// TwinCAT 3 PLC project Fraktal_Press_Demo
// Title: Fraktal_Press_Demo
// Company: fraktal-automation
// Author: fraktal-automation
// ProjectVersion: 0.1.0.7
// Description: CX2030 virtual/physical commissioning example: XTI-linked EK1200/EL1809/EL2809 HAL mapping, two-hand start, interlocked door/part slide, safety aliases, Control On/Off, AUTO/HOME/MANUAL, and model recipes.
// ProgramVersion: 3.1.4024.0
// libraries:
//   Tc2_Standard, * (Beckhoff Automation GmbH)
//   Tc3_Module, * (Beckhoff Automation GmbH)
//   Fraktal_Core, 0.1.0.3 (fraktal-automation)
//   Fraktal_Modules, 0.1.0.2 (fraktal-automation)
// project tree:
//   / PlcTask.TcTTO
//   01_PneumaticPress/Sequences/ FB_PressDemoLoadPosition.TcPOU, FB_PressDemoHome.TcPOU, FB_PressDemoChangeover.TcPOU, FB_PressDemoAuto.TcPOU
//   01_PneumaticPress/Release/ FB_PressDemoRelease.TcPOU
//   01_PneumaticPress/ FB_PressDemoUnit.TcPOU
//   00_System/ MAIN.TcPOU, GVL_PressIO.TcGVL, GVL_PressSafety.TcGVL, FB_PressIoDriver.TcPOU, FB_PressControlDomain.TcPOU, FB_PressOutputAuthority.TcPOU, FB_PressSimulationDriver.TcPOU
//   01_PneumaticPress/Recipes/ FB_PressRecipeCatalog.TcPOU
//   01_PneumaticPress/Io/ FB_PressIoCatalog.TcPOU, GVL_PressFieldbus.TcGVL

CONFIGURATION Fraktal_Press_Demo
    RESOURCE PLC ON TwinCAT3
        TASK PlcTask(INTERVAL := T#10ms, PRIORITY := 20);
        PROGRAM MAIN WITH PlcTask : MAIN;
    END_RESOURCE
END_CONFIGURATION

// ---- 00_System/GVL_PressIO.TcGVL
{attribute 'qualified_only'}
// CX2030 local EtherCAT process image, reconciled with the supplied XTI export.
// TcLinkTo owns the physical link by exact terminal/channel/PDO-entry name;
// AT %I*/%Q* keeps the compiler-selected process-image offset non-positional.
VAR_GLOBAL
    // =000+S-K010B1 (EL1809) inputs
    {attribute 'TcLinkTo' := 'TIIB[=000+S-K010B1 (EL1809)]^Channel 1^_101B301A'}
    _101B301A AT %I* : BOOL;       // Ch1 feeder retracted = logical slide INSIDE
    {attribute 'TcLinkTo' := 'TIIB[=000+S-K010B1 (EL1809)]^Channel 2^_101B301B'}
    _101B301B AT %I* : BOOL;       // Ch2 feeder extended  = logical slide OUTSIDE
    {attribute 'TcLinkTo' := 'TIIB[=000+S-K010B1 (EL1809)]^Channel 3^_101B201A'}
    _101B201A AT %I* : BOOL;       // Ch3 door closed
    {attribute 'TcLinkTo' := 'TIIB[=000+S-K010B1 (EL1809)]^Channel 4^_101B201B'}
    _101B201B AT %I* : BOOL;       // Ch4 door open
    {attribute 'TcLinkTo' := 'TIIB[=000+S-K010B1 (EL1809)]^Channel 5^_101B202A'}
    _101B202A AT %I* : BOOL;       // Ch5 press down
    {attribute 'TcLinkTo' := 'TIIB[=000+S-K010B1 (EL1809)]^Channel 6^_101B202B'}
    _101B202B AT %I* : BOOL;       // Ch6 press up
    {attribute 'TcLinkTo' := 'TIIB[=000+S-K010B1 (EL1809)]^Channel 7^_101S101'}
    _101S101  AT %I* : BOOL;       // Ch7 right two-hand raw button
    {attribute 'TcLinkTo' := 'TIIB[=000+S-K010B1 (EL1809)]^Channel 8^_101S102'}
    _101S102  AT %I* : BOOL;       // Ch8 left two-hand raw button
    {attribute 'TcLinkTo' := 'TIIB[=000+S-K010B1 (EL1809)]^Channel 10^_000MB085A_2'}
    _000MB085A_2 AT %I* : BOOL;    // Ch10 compressed air below 0.3 bar
    {attribute 'TcLinkTo' := 'TIIB[=000+S-K010B1 (EL1809)]^Channel 11^_000MB085A_4'}
    _000MB085A_4 AT %I* : BOOL;    // Ch11 compressed air above 4.5 bar
    {attribute 'TcLinkTo' := 'TIIB[=000+S-K010B1 (EL1809)]^Channel 12^_101B601'}
    _101B601 AT %I* : BOOL;        // Ch12 part present
    {attribute 'TcLinkTo' := 'TIIB[=000+S-K010B1 (EL1809)]^Channel 14^_000K911_Y32'}
    _000K911_Y32 AT %I* : BOOL;    // Ch14 Control On feedback
    {attribute 'TcLinkTo' := 'TIIB[=000+S-K010B1 (EL1809)]^Channel 15^_000K910A'}
    _000K910A AT %I* : BOOL;       // Ch15 ordinary E-stop healthy mirror only

    // =000+S-K010C1 (EL2809) outputs
    {attribute 'TcLinkTo' := 'TIIB[=000+S-K010C1 (EL2809)]^Channel 1^_101K301A'}
    _101K301A AT %Q* : BOOL;       // Ch1 feeder backward = move inside
    {attribute 'TcLinkTo' := 'TIIB[=000+S-K010C1 (EL2809)]^Channel 2^_101K301B'}
    _101K301B AT %Q* : BOOL;       // Ch2 feeder forward  = move outside
    {attribute 'TcLinkTo' := 'TIIB[=000+S-K010C1 (EL2809)]^Channel 3^_101K201A'}
    _101K201A AT %Q* : BOOL;       // Ch3 close door
    {attribute 'TcLinkTo' := 'TIIB[=000+S-K010C1 (EL2809)]^Channel 4^_101K201B'}
    _101K201B AT %Q* : BOOL;       // Ch4 open door
    {attribute 'TcLinkTo' := 'TIIB[=000+S-K010C1 (EL2809)]^Channel 5^_101K202A'}
    _101K202A AT %Q* : BOOL;       // Ch5 press downward
    {attribute 'TcLinkTo' := 'TIIB[=000+S-K010C1 (EL2809)]^Channel 6^_101K202B'}
    _101K202B AT %Q* : BOOL;       // Ch6 press upward
    {attribute 'TcLinkTo' := 'TIIB[=000+S-K010C1 (EL2809)]^Channel 7^_101P101'}
    _101P101  AT %Q* : BOOL;       // Ch7 right two-hand lamp
    {attribute 'TcLinkTo' := 'TIIB[=000+S-K010C1 (EL2809)]^Channel 8^_101P102'}
    _101P102  AT %Q* : BOOL;       // Ch8 left two-hand lamp
    {attribute 'TcLinkTo' := 'TIIB[=000+S-K010C1 (EL2809)]^Channel 10^_000K951_A1'}
    _000K951_A1 AT %Q* : BOOL;     // Ch10 SwitchControlOn functional request
    {attribute 'TcLinkTo' := 'TIIB[=000+S-K010C1 (EL2809)]^Channel 11^_000K911_A1'}
    _000K911_A1 AT %Q* : BOOL;     // Ch11 EnableControlOn functional request
END_VAR

// ---- 00_System/GVL_PressSafety.TcGVL
{attribute 'qualified_only'}
// Read-only aliases to results produced outside the standard PLC by TwinSAFE
// or a validated external safety system. They intentionally default FALSE so
// physical mode cannot energize until commissioning supplies every result.
// These variables do not themselves implement a safety function.
VAR_GLOBAL
    _EStopOk               AT %I* : BOOL;
    _GuardClosed           AT %I* : BOOL;
    _TwoHandActive         AT %I* : BOOL;
    _PneumaticPermit       AT %I* : BOOL;
    _SafetyFieldbusHealthy AT %I* : BOOL;
    _StandardIoHealthy     AT %I* : BOOL;
END_VAR

// ---- 01_PneumaticPress/Io/GVL_PressFieldbus.TcGVL
{attribute 'qualified_only'}
{attribute 'OPC.UA.DA' := '1'}
// Owner-local, bounded publication of the demo's physical CX2030 I/O tree.
// ST_IoChannel.Name is always the exact electrical-list/schematic tag.
VAR_GLOBAL
    Topology : ST_FieldbusTopology;
END_VAR

// ---- 00_System/MAIN.TcPOU
// Virtual-commissioning application for one pneumatic press Unit.
// IMPORTANT: the Safe* values below simulate TwinSAFE outputs only. A deployed
// machine maps certified E-stop/two-hand/guard/safe-valve results from TwinSAFE.
PROGRAM MAIN
VAR
    RecipeCatalog : FB_PressRecipeCatalog;
    PartCarrier : FB_LocalPartCarrier;    // §3.16.2 BY_POSITION identity + local result ring
    AccessUsers : FB_LocalAccessProvider; // §7.7 commissioning user/PIN table
    // TF6100 TMC-Filtered publication starts at the deployed root instance.
    // The marker is inherited by PneumaticPress's published child symbols.
    {attribute 'OPC.UA.DA' := '1'}
    PneumaticPress : FB_PressDemoUnit;
    IoCatalog : FB_PressIoCatalog;
    IoDriver : FB_PressIoDriver;
    ControlDomain : FB_PressControlDomain;
    OutputAuthority : FB_PressOutputAuthority;
    SimulationDriver : FB_PressSimulationDriver;
    PressHal, DoorHal, SlideHal : ST_CylinderHal;
    TwoHandHal : ST_TwoHandHal;
    PowerHal : ST_PowerGroupHal;
    PartPresentHal : ST_DigitalInputHal;
    AirPressureHal : ST_AirPressureHal;
    InitialModel : ST_ModelId;
    Plate : ST_Nameplate;
    Init : BOOL;
    UseSimulation : BOOL := TRUE; // set FALSE only after I/O + safety aliases are linked
    ControlCircuitMappingConfirmed : BOOL; // verify K951/K911 electrical semantics first

    // Simulation controls. E-stop is normally closed: TRUE = healthy circuit.
    SimEStopNc : BOOL := TRUE;
    SimControlOnButton : BOOL;
    SimControlOffButton : BOOL;
    SimLeftButton : BOOL;
    SimRightButton : BOOL;
    SimSafetyValveOk : BOOL := TRUE;
    SimFieldbusHealthy : BOOL := TRUE;
    SimPartPresent : BOOL := TRUE;
    SimAirPressureOk : BOOL := TRUE;
    SafeEStopOk : BOOL;
    SafeGuardClosed : BOOL;
    SafeTwoHandActive : BOOL;
    SafePneumaticPermit : BOOL;
    SafetyFieldbusHealthy : BOOL;
    StandardIoHealthy : BOOL;
    RawEStopHealthy : BOOL;
    LampsOn : BOOL;
    ControlOnEdge : R_TRIG;
    ControlOffEdge : R_TRIG;
END_VAR

IF NOT Init THEN
    Init := TRUE;
    // Initial mechanically safe/load position: ram up, door open, slide outside.
    PressHal.RetractedFb := TRUE;
    DoorHal.RetractedFb := TRUE;
    SlideHal.RetractedFb := TRUE;
    RecipeCatalog.Setup(UnitRef := PneumaticPress);
    PneumaticPress.Setup(Name := 'PneumaticPress', PressHal := PressHal, DoorHal := DoorHal,
        SlideHal := SlideHal, TwoHandHal := TwoHandHal, PowerHal := PowerHal,
        PartPresentHal := PartPresentHal, AirPressureHal := AirPressureHal,
        Recipe := RecipeCatalog.Provider);
    IoDriver.Setup(UnitRef := PneumaticPress);
    IoCatalog.Setup(UnitRef := PneumaticPress);
    ControlDomain.Setup(UnitRef := PneumaticPress);
    SimulationDriver.Setup(PressHal := PressHal, DoorHal := DoorHal, SlideHal := SlideHal);
    InitialModel.ModelCode := 'ALUMINUM';
    PneumaticPress.SetModel(Id := InitialModel);
    Plate.ProductUri := 'urn:fraktal:demo:pneumatic-press:2026-0001';
    Plate.ManufacturerName := 'Fraktal Example Project';
    Plate.ProductDesignation := 'Pneumatic Press Training Cell';
    Plate.SerialNumber := 'PRESS-DEMO-2026-0001';
    Plate.YearOfConstruction := '2026';
    Plate.SoftwareVersion := 'Fraktal Press Demo 0.1';
    PneumaticPress.SetNameplate(Plate := Plate);
    PneumaticPress.AlarmLog.RegisterMeta(Reason := E_Reason.INTERLOCK_DROPPED,
        OperatorAction := 'project.alarmAction.pressInterlock',
        Consequence := 'project.alarmConsequence.pressInterlock', Shelvable := FALSE);
    // §8.9 rationalization: per-reason operator action + consequence for the HMI join
    PneumaticPress.AlarmLog.RegisterMeta(Reason := E_Reason.PERMISSIVE_NOT_MET,
        OperatorAction := 'project.alarmAction.pressAirPressure',
        Consequence := 'project.alarmConsequence.pressAirPressure', Shelvable := FALSE);
    PneumaticPress.AlarmLog.RegisterMeta(Reason := E_Reason.RECIPE_INVALID,
        OperatorAction := 'project.alarmAction.pressRecipe',
        Consequence := 'project.alarmConsequence.pressRecipe', Shelvable := FALSE);
    PneumaticPress.AlarmLog.RegisterMeta(Reason := PL_ModuleReasons.CYL_WORK_NOT_REACHED,
        OperatorAction := 'project.alarmAction.pressCylinderPosition',
        Consequence := 'project.alarmConsequence.pressCylinderPosition', Shelvable := FALSE);
    PneumaticPress.AlarmLog.RegisterMeta(Reason := PL_ModuleReasons.CYL_HOME_NOT_REACHED,
        OperatorAction := 'project.alarmAction.pressCylinderPosition',
        Consequence := 'project.alarmConsequence.pressCylinderPosition', Shelvable := FALSE);
    // §3.16 traceability: station-local BY_POSITION serials; RFID/host substitutes later
    PartCarrier.Setup(UidPrefix := 'PRESS-2026-');
    PneumaticPress.SetPartCarrier(Carrier := PartCarrier);
    // §7.7 access: commissioning users (policy stays shipped-open; login is optional)
    AccessUsers.Register(User := 'operator', Pin := '1111', Level := E_AccessLevel.OPERATOR);
    AccessUsers.Register(User := 'tech', Pin := '2222', Level := E_AccessLevel.TECHNICIAN);
    AccessUsers.Register(User := 'admin', Pin := '9999', Level := E_AccessLevel.ADMIN);
    PneumaticPress.Access.Setup(Provider := AccessUsers, pAlarmLog := ADR(PneumaticPress.AlarmLog));
END_IF

// Ordinary simulated local station buttons. The worksheet does not list real
// Control On/Off input buttons; physical operation therefore uses HMI requests
// until those devices are identified. Control Off wins simultaneous edges.
ControlOnEdge(CLK := UseSimulation AND SimControlOnButton);
ControlOffEdge(CLK := UseSimulation AND SimControlOffButton);
IF ControlOffEdge.Q THEN
    PneumaticPress.RequestLocalControl(ControlOn := FALSE);
ELSIF ControlOnEdge.Q THEN
    PneumaticPress.RequestLocalControl(ControlOn := TRUE);
END_IF

IF UseSimulation THEN
    SimulationDriver.M_ReadInputs(DoorHal := DoorHal, TwoHandHal := TwoHandHal,
        PowerHal := PowerHal, PartPresentHal := PartPresentHal,
        AirPressureHal := AirPressureHal, RawEStopHealthy := RawEStopHealthy,
        SafeEStopOk := SafeEStopOk, SafeGuardClosed := SafeGuardClosed,
        SafeTwoHandActive := SafeTwoHandActive,
        SafePneumaticPermit := SafePneumaticPermit,
        SafetyFieldbusHealthy := SafetyFieldbusHealthy,
        StandardIoHealthy := StandardIoHealthy, SimEStopNc := SimEStopNc,
        SimLeftButton := SimLeftButton, SimRightButton := SimRightButton,
        SimSafetyValveOk := SimSafetyValveOk,
        SimFieldbusHealthy := SimFieldbusHealthy,
        SimPartPresent := SimPartPresent, SimAirPressureOk := SimAirPressureOk,
        PowerRequested := PowerHal.EnableRequestOut);
ELSE
    // The project Hardware Driver is the only raw process-image consumer.
    IoDriver.M_ReadInputs(PressHal := PressHal, DoorHal := DoorHal,
        SlideHal := SlideHal, TwoHandHal := TwoHandHal, PowerHal := PowerHal,
        PartPresentHal := PartPresentHal, AirPressureHal := AirPressureHal,
        RawEStopHealthy := RawEStopHealthy, SafeEStopOk := SafeEStopOk,
        SafeGuardClosed := SafeGuardClosed, SafeTwoHandActive := SafeTwoHandActive,
        SafePneumaticPermit := SafePneumaticPermit,
        SafetyFieldbusHealthy := SafetyFieldbusHealthy,
        StandardIoHealthy := StandardIoHealthy);
END_IF
TwoHandHal.SafeActive := SafeTwoHandActive;
TwoHandHal.FieldbusHealthy := SafetyFieldbusHealthy;
PowerHal.SafetyPermit := SafePneumaticPermit;
PowerHal.FieldbusHealthy := StandardIoHealthy;

ControlDomain.M_Update(SafeEStopOk := SafeEStopOk,
    SafeGuardClosed := SafeGuardClosed, SafeTwoHandActive := SafeTwoHandActive,
    SafePneumaticPermit := SafePneumaticPermit,
    SafetyFieldbusHealthy := SafetyFieldbusHealthy,
    StandardIoHealthy := StandardIoHealthy, RawEStopHealthy := RawEStopHealthy,
    PowerFeedback := PowerHal.PowerFeedback,
    PowerRequested := PowerHal.EnableRequestOut,
    TwoHandFieldbusHealthy := TwoHandHal.FieldbusHealthy);
PneumaticPress.ControlDomain := ControlDomain.Status;

// First execute ordinary control, then apply a standard-PLC withdrawal layer.
// This is defense in depth only: the real safety system owns pneumatic removal.
PneumaticPress();
OutputAuthority.M_Apply(PressHal := PressHal, DoorHal := DoorHal,
    SlideHal := SlideHal, PowerFeedback := PowerHal.PowerFeedback,
    SafePneumaticPermit := SafePneumaticPermit,
    StandardIoHealthy := StandardIoHealthy,
    HazardousRamPermit := SafeGuardClosed AND SafeTwoHandActive);
IF UseSimulation THEN
    // Never leave physical outputs energized while virtual commissioning.
    IoDriver.M_ClearOutputs();
    SimulationDriver.M_RefreshPlant();
ELSE
    LampsOn := PneumaticPress.TwoHand.OutImm.Armed
        AND ControlDomain.Status.ReadyForStart
        AND PneumaticPress.OutImm.PartPresent AND PneumaticPress.OutImm.AirPressureOk;
    IoDriver.M_WriteOutputs(PressHal := PressHal, DoorHal := DoorHal,
        SlideHal := SlideHal, PowerHal := PowerHal, LampsOn := LampsOn,
        ControlCircuitMappingConfirmed := ControlCircuitMappingConfirmed);
END_IF
IoDriver.M_RefreshFieldbus(StandardIoHealthy := StandardIoHealthy);

END_PROGRAM

// ---- 01_PneumaticPress/Recipes/FB_PressRecipeCatalog.TcPOU
// Owner-local recipe engineering data: model identities and their typed Unit records.
// Generic validation/storage remains in FB_LocalRecipeProvider; process behavior
// remains in the project-owned FB_PressDemoUnit. MAIN only composes the two.
FUNCTION_BLOCK FB_PressRecipeCatalog
VAR_OUTPUT
    {attribute 'OPC.UA.DA' := '0'}
    Provider : FB_LocalRecipeProvider;
END_VAR
VAR
    _default : ST_PneumaticPressParCfg;
    _aluminum : ST_PneumaticPressParCfg;
    _plastic : ST_PneumaticPressParCfg;
    _steel : ST_PneumaticPressParCfg;
    _model : ST_ModelId;
    _configured : BOOL;
END_VAR

// Static catalog: no cyclic work.

METHOD Setup : BOOL
VAR_INPUT
    UnitRef : REFERENCE TO FB_PressDemoUnit;
END_VAR
VAR
    Ok : BOOL;
END_VAR
IF _configured THEN
    Setup := TRUE;
    RETURN;
END_IF

// §8.11 per-model performance references: IdealCycleMs feeds OEE Performance
// (§8.5.1); BaselineWorkMs arms the WORK-time degradation watch (§8.11.4(d)).
// Values = design cycle for this training cell (motions + settle + dwell).
_default.PressSettleTime := T#500MS;
_default.TransferSettleTime := T#100MS;
_default.RequireTwoHandStart := TRUE;
_default.IdealCycleMs := 6000;
_default.BaselineWorkMs := 6000;
_aluminum.PressSettleTime := T#300MS;
_aluminum.TransferSettleTime := T#80MS;
_aluminum.RequireTwoHandStart := TRUE;
_aluminum.IdealCycleMs := 5700;
_aluminum.BaselineWorkMs := 5700;
_plastic.PressSettleTime := T#650MS;
_plastic.TransferSettleTime := T#120MS;
_plastic.RequireTwoHandStart := TRUE;
_plastic.IdealCycleMs := 6200;
_plastic.BaselineWorkMs := 6200;
_steel.PressSettleTime := T#1200MS;
_steel.TransferSettleTime := T#150MS;
_steel.RequireTwoHandStart := TRUE;
_steel.IdealCycleMs := 6800;
_steel.BaselineWorkMs := 6800;

Ok := Provider.Register(ModelCode := '', RecipeKey := 'PneumaticPressUnit',
    pData := ADR(_default), Size := SIZEOF(_default));
Ok := Provider.Register(ModelCode := 'ALUMINUM', RecipeKey := 'PneumaticPressUnit',
    pData := ADR(_aluminum), Size := SIZEOF(_aluminum)) AND Ok;
Ok := Provider.Register(ModelCode := 'PLASTIC', RecipeKey := 'PneumaticPressUnit',
    pData := ADR(_plastic), Size := SIZEOF(_plastic)) AND Ok;
Ok := Provider.Register(ModelCode := 'STEEL', RecipeKey := 'PneumaticPressUnit',
    pData := ADR(_steel), Size := SIZEOF(_steel)) AND Ok;

_model.ModelCode := 'ALUMINUM';
Ok := UnitRef.RegisterAvailableModel(Id := _model) AND Ok;
_model.ModelCode := 'PLASTIC';
Ok := UnitRef.RegisterAvailableModel(Id := _model) AND Ok;
_model.ModelCode := 'STEEL';
Ok := UnitRef.RegisterAvailableModel(Id := _model) AND Ok;

_configured := Ok;
Setup := Ok;
END_METHOD

END_FUNCTION_BLOCK

// ---- 01_PneumaticPress/FB_PressDemoUnit.TcPOU
// Project-owned Unit: pneumatic press + access door + transfer slide + two-hand request.
// Cylinder interlocks prevent the two documented collisions in AUTO and MANUAL.
// Certified E-stop, two-hand evaluation and safe valve outputs remain external.
{attribute 'OPC.UA.DA' := '1'}
FUNCTION_BLOCK FB_PressDemoUnit EXTENDS FB_UnitBase
VAR_INPUT
    ParCfg : ST_PneumaticPressParCfg;
    ParCmd : ST_PneumaticPressParCmd;
END_VAR
VAR_OUTPUT
    PressRam      : FB_CylinderCM;
    Door          : FB_CylinderCM;
    PartSlide     : FB_CylinderCM;
    TwoHand       : FB_TwoHandStartCM;
    PneumaticPower: FB_PowerGroupCM;
    PartPresentSensor : FB_DigitalInputCM;
    AirPressureMonitor : FB_AirPressureMonitorCM;
    ReleaseConditions : FB_PressDemoRelease; // project-owned, browseable condition state
    OutCmd        : ST_PneumaticPressOutCmd;
    OutImm        : ST_PneumaticPressOutImm;
END_VAR
VAR
    _recipe : I_RecipeProvider;
    _parCfgStaged : ST_PneumaticPressParCfg;
    _recipePrepared : BOOL;
    _startLatched : BOOL;
    _powerRequestPending : BOOL;
    _powerTargetOn : BOOL;
    {attribute 'OPC.UA.DA' := '0'}
    _homeSequence : FB_PressDemoHome;       // §6.8 ST chain on FB_SequenceBase owns HOME steps
    {attribute 'OPC.UA.DA' := '0'}
    _changeoverSequence : FB_PressDemoChangeover;
    {attribute 'OPC.UA.DA' := '0'}
    _autoSequence : FB_PressDemoAuto;
END_VAR

Cyclic();

METHOD Setup : BOOL
VAR_INPUT
    Name : STRING(80);
    PressHal : REFERENCE TO ST_CylinderHal;
    DoorHal : REFERENCE TO ST_CylinderHal;
    SlideHal : REFERENCE TO ST_CylinderHal;
    TwoHandHal : REFERENCE TO ST_TwoHandHal;
    PowerHal : REFERENCE TO ST_PowerGroupHal;
    PartPresentHal : REFERENCE TO ST_DigitalInputHal;
    AirPressureHal : REFERENCE TO ST_AirPressureHal;
    Recipe : I_RecipeProvider;
END_VAR
VAR
    InitialModel : ST_ModelId;
    Ok : BOOL;
END_VAR
_M_SetName(Name);
_M_SetPresentation(DisplayNameKey := 'project.module.pneumaticPress.name', DescriptionKey := 'project.module.pneumaticPress.description');
_recipe := Recipe;
Ok := PressRam.Setup(Name := CONCAT(Name, '.PressRam'), HalRef := PressHal, Recipe := 0);
Ok := Door.Setup(Name := CONCAT(Name, '.Door'), HalRef := DoorHal, Recipe := 0) AND Ok;
Ok := PartSlide.Setup(Name := CONCAT(Name, '.PartSlide'), HalRef := SlideHal, Recipe := 0) AND Ok;
Ok := TwoHand.Setup(Name := CONCAT(Name, '.TwoHand'), HalRef := TwoHandHal) AND Ok;
Ok := PneumaticPower.Setup(Name := CONCAT(Name, '.PneumaticPower'), HalRef := PowerHal) AND Ok;
Ok := PartPresentSensor.Setup(Name := CONCAT(Name, '.PartPresentSensor'),
    HalRef := PartPresentHal, DisplayNameKey := 'project.module.partPresentSensor.name',
    DescriptionKey := 'project.module.partPresentSensor.description') AND Ok;
Ok := AirPressureMonitor.Setup(Name := CONCAT(Name, '.AirPressureMonitor'),
    HalRef := AirPressureHal) AND Ok;
Ok := ReleaseConditions.Setup(UnitPath := Name) AND Ok;
Ok := _homeSequence.Setup(Host := THIS^, PressRam := PressRam, Door := Door,
    PartSlide := PartSlide, OutCmd := OutCmd) AND Ok;
Ok := _changeoverSequence.Setup(Host := THIS^, PressRam := PressRam, Door := Door,
    PartSlide := PartSlide, OutCmd := OutCmd, Model := Model) AND Ok;
Ok := _autoSequence.Setup(Host := THIS^, PressRam := PressRam, Door := Door,
    PartSlide := PartSlide, TwoHand := TwoHand, PartPresentSensor := PartPresentSensor,
    AirPressureMonitor := AirPressureMonitor, ParCfg := ParCfg, OutCmd := OutCmd,
    StartLatched := _startLatched) AND Ok;
PneumaticPower.ParCfg.Kind := E_PowerGroupKind.VALVE_ZONE;
PneumaticPower.ParCfg.RequiredForControl := TRUE;
PneumaticPower.ParCfg.FieldbusLossReaction := E_FieldbusLossReaction.CONTROL_OFF;
Ok := _M_Register(PressRam) AND Ok;
Ok := _M_Register(Door) AND Ok;
Ok := _M_Register(PartSlide) AND Ok;
Ok := _M_Register(TwoHand) AND Ok;
Ok := _M_Register(PneumaticPower) AND Ok;
Ok := _M_Register(PartPresentSensor) AND Ok;
Ok := _M_Register(AirPressureMonitor) AND Ok;
Setup := Ok AND PrepareRecipe(Model := InitialModel);
IF Setup THEN CommitRecipe(); END_IF
END_METHOD

METHOD PrepareRecipe : BOOL
VAR_INPUT
    Model : ST_ModelId;
END_VAR
IF _recipe = 0 THEN
    _parCfgStaged := ParCfg;
    _recipePrepared := TRUE;
ELSIF _recipe.Load(ModelCode := Model.ModelCode, RecipeKey := 'PneumaticPressUnit', pParCfg := ADR(_parCfgStaged), Size := SIZEOF(_parCfgStaged)) THEN
    IF (_parCfgStaged.PressSettleTime > T#30S) OR (_parCfgStaged.TransferSettleTime > T#5S) THEN
        _M_Fault(E_Reason.RECIPE_INVALID, 'project.error.pressRecipeInvalid');
        _recipePrepared := FALSE;
        PrepareRecipe := FALSE;
        RETURN;
    END_IF
    _recipePrepared := TRUE;
ELSE
    _M_Fault(E_Reason.RECIPE_INVALID, 'std.error.recipeSchemaInvalid');
    _recipePrepared := FALSE;
    PrepareRecipe := FALSE;
    RETURN;
END_IF
PrepareRecipe := SUPER^.PrepareRecipe(Model := Model);
IF NOT PrepareRecipe THEN _recipePrepared := FALSE; END_IF
END_METHOD

METHOD CommitRecipe
SUPER^.CommitRecipe();
IF _recipePrepared THEN
    ParCfg := _parCfgStaged;
    // §8.11 performance references follow the model: OEE Performance denominator
    // and the WORK-time degradation baseline are per-recipe engineering data.
    Oee.IdealCycleMs := ParCfg.IdealCycleMs;
    Profiler.M_SetBaselineWork(WorkMs := ParCfg.BaselineWorkMs);
END_IF
_recipePrepared := FALSE;
END_METHOD

METHOD AbortRecipe
SUPER^.AbortRecipe();
_recipePrepared := FALSE;
END_METHOD

METHOD PROTECTED OnCyclic : DINT
OnCyclic := SUPER^.OnCyclic();
// Project release engineering is a separate visible component. It owns the
// functional collision permits and mode-entry conditions consumed below.
ReleaseConditions.M_Evaluate(PressRam := PressRam, Door := Door, PartSlide := PartSlide,
    TwoHand := TwoHand, PneumaticPower := PneumaticPower,
    AirPressure := AirPressureMonitor);

// Latch access-gated Unit requests, then observe one full Execute-low scan before
// starting another power-group command (PLCopen edge discipline).
IF ControlOffRequest THEN
    _powerTargetOn := FALSE;
    _powerRequestPending := TRUE;
ELSIF ControlOnRequest THEN
    _powerTargetOn := TRUE;
    _powerRequestPending := TRUE;
END_IF
IF PneumaticPower.Done OR PneumaticPower.Error OR PneumaticPower.Aborted THEN
    PneumaticPower.Execute := FALSE;
ELSIF _powerRequestPending AND NOT PneumaticPower.Execute
AND (PneumaticPower.State = E_ExecState.READY) THEN
    PneumaticPower.Abort := FALSE;
    IF _powerTargetOn THEN
        PneumaticPower.Command := E_PowerGroupCommand.POWER_ON;
    ELSE
        PneumaticPower.Command := E_PowerGroupCommand.POWER_OFF;
    END_IF
    PneumaticPower.Execute := TRUE;
    _powerRequestPending := FALSE;
END_IF

// A physical two-hand edge may start AUTO from READY, or release an already
// running Unit's wait step. It never bypasses domain readiness or access policy.
IF TwoHand.OutImm.StartPulse
AND PartPresentSensor.OutImm.Value AND PartPresentSensor.OutImm.Quality
AND AirPressureMonitor.OutImm.PressureOk THEN
    IF (State = E_ExecState.BUSY) AND (ModeActive = E_Mode.AUTO) THEN
        _startLatched := TRUE;
    ELSIF (ModeActive = E_Mode.AUTO) AND Start() THEN
        _startLatched := TRUE;
    END_IF
ELSIF TwoHand.OutImm.StartPulse THEN
    _startLatched := FALSE;
END_IF
IF PneumaticPower.Error AND (State = E_ExecState.BUSY) THEN
    _M_RollupFault();
END_IF
IF (State = E_ExecState.BUSY) AND (_step > 10)
AND NOT AirPressureMonitor.OutImm.PressureOk THEN
    PressRam.WithdrawOutputs();
    Door.WithdrawOutputs();
    PartSlide.WithdrawOutputs();
    _M_Fault(E_Reason.PERMISSIVE_NOT_MET, 'project.error.pressAirPressureLost');
END_IF
OutImm.PressRetracted := PressRam.OutImm.Retracted;
OutImm.DoorOpen := Door.OutImm.Retracted;
OutImm.DoorClosed := Door.OutImm.Extended;
OutImm.SlideInside := PartSlide.OutImm.Extended;
OutImm.SlideOutside := PartSlide.OutImm.Retracted;
OutImm.TwoHandArmed := TwoHand.OutImm.Armed;
OutImm.TwoHandActive := TwoHand.OutImm.SafeActive;
OutImm.PartPresent := PartPresentSensor.OutImm.Value AND PartPresentSensor.OutImm.Quality;
OutImm.AirPressureOk := AirPressureMonitor.OutImm.PressureOk;
OutImm.ReadyForLoad := Door.OutImm.Retracted AND NOT Door.OutImm.Extended
    AND PartSlide.OutImm.Retracted AND NOT PartSlide.OutImm.Extended
    AND PressRam.OutImm.Retracted AND NOT PressRam.OutImm.Extended;
OutImm.ActiveSettleTime := ParCfg.PressSettleTime;
OutImm.Diagnostic := Status.Diagnostic;
END_METHOD

METHOD PROTECTED OnAbort : DINT
OnAbort := SUPER^.OnAbort();
_M_PartAborted();                    // §3.16.3: the part leaves without a valid result
PressRam.WithdrawOutputs();
Door.WithdrawOutputs();
PartSlide.WithdrawOutputs();
PressRam.Execute := FALSE;
Door.Execute := FALSE;
PartSlide.Execute := FALSE;
Decision.Prompt := '';
DecisionAnswer := 0;
_startLatched := FALSE;
_homeSequence.M_Reset();
_changeoverSequence.M_Reset();
_autoSequence.M_Reset();
_powerTargetOn := FALSE;
_powerRequestPending := TRUE;
END_METHOD

// Application-only seam for ordinary hardwired Control On/Off buttons.
// It is a method (not OPC UA data), so HMI writes still use the access-gated
// ReqControlOn/ReqControlOff contract. The power CM rechecks safety and health.
METHOD RequestLocalControl : BOOL
VAR_INPUT
    ControlOn : BOOL;
END_VAR
_powerTargetOn := ControlOn;
_powerRequestPending := TRUE;
RequestLocalControl := TRUE;
END_METHOD

// §3.4.2 — the press paces every motion boundary through _M_StepGate, so
// SINGLE_STEP and HOLD_TO_RUN are supported (NON-SAFETY pacing; interlocks
// and the certified safety layer are unaffected).
METHOD PROTECTED _M_SupportsRunStyle : BOOL
VAR_INPUT
    Style : E_RunStyle;
END_VAR
_M_SupportsRunStyle := (Style = E_RunStyle.CONTINUOUS)
    OR (Style = E_RunStyle.SINGLE_STEP) OR (Style = E_RunStyle.HOLD_TO_RUN);
END_METHOD

METHOD PROTECTED _M_Supports : BOOL
VAR_INPUT
    Mode : E_Mode;
END_VAR
_M_Supports := (Mode = E_Mode.AUTO) OR (Mode = E_Mode.MANUAL)
    OR (Mode = E_Mode.HOME) OR (Mode = E_Mode.CHANGEOVER);
END_METHOD

// Thin mode router. Each supported sequence is a named method in the Unit tree.
METHOD PROTECTED _M_Dispatch
CASE ModeActive OF
    E_Mode.AUTO:
        _M_SequenceAuto();
    E_Mode.HOME:
        _M_SequenceHome();
    E_Mode.CHANGEOVER:
        _M_SequenceChangeover();
    E_Mode.MANUAL:
        _M_Fault(E_Reason.UNSUPPORTED_COMMAND, 'project.error.pressManualHasNoSequence');
ELSE
    _M_Fault(E_Reason.UNSUPPORTED_COMMAND, 'project.error.pressModeHasNoSequence');
END_CASE
END_METHOD

// HOME adapter: reset the chain on the first dispatch scan, then run it each scan.
// The §6.8 ST chain (FB_PressDemoHome) owns all HOME step logic.
METHOD PROTECTED _M_SequenceHome
CASE _step OF
    10:
        _homeSequence.M_Reset();
        _step := 20;
    20:
        _homeSequence.M_Run();
ELSE
    PressRam.WithdrawOutputs();
    Door.WithdrawOutputs();
    PartSlide.WithdrawOutputs();
    _M_Fault(E_Reason.STEP_STALLED, 'std.error.undefinedStep');
END_CASE
END_METHOD

// CHANGEOVER adapter: reset then run. The §6.8 ST chain owns model validation,
// safe positioning, the operator decision, and completion logic.
METHOD PROTECTED _M_SequenceChangeover
CASE _step OF
    10:
        _changeoverSequence.M_Reset();
        _step := 20;
    20:
        _changeoverSequence.M_Run();
ELSE
    PressRam.WithdrawOutputs();
    Door.WithdrawOutputs();
    PartSlide.WithdrawOutputs();
    _M_Fault(E_Reason.STEP_STALLED, 'std.error.undefinedStep');
END_CASE
END_METHOD

// AUTO adapter: reset then run. Every production step's command, wait, timer,
// decision, traceability, and transition logic lives in the §6.8 ST chain.
METHOD PROTECTED _M_SequenceAuto
CASE _step OF
    10:
        _autoSequence.M_Reset();
        _step := 20;
    20:
        _autoSequence.M_Run();
ELSE
    PressRam.WithdrawOutputs();
    Door.WithdrawOutputs();
    PartSlide.WithdrawOutputs();
    _M_Fault(E_Reason.STEP_STALLED, 'std.error.undefinedStep');
END_CASE
END_METHOD

METHOD PROTECTED _M_RouteManual : BOOL
VAR_INPUT
    TargetPath : STRING(255);
    Value : DINT;
END_VAR
_M_RouteManual := FALSE;
IF TargetPath = PressRam.Name THEN
    _M_RouteManual := PressRam.ManualCommand(Value := Value);
ELSIF TargetPath = Door.Name THEN
    _M_RouteManual := Door.ManualCommand(Value := Value);
ELSIF TargetPath = PartSlide.Name THEN
    _M_RouteManual := PartSlide.ManualCommand(Value := Value);
ELSE
    _M_RouteManual := FALSE;
END_IF
END_METHOD

// §7.8 mode-entry release owned by this Unit. The base Start method consumes the
// same report the HMI displays, so this condition cannot become explanation-only.
METHOD PROTECTED _M_AppendInterlocks
VAR_IN_OUT
    Report : ST_ReleaseReport;
END_VAR
ReleaseConditions.M_AppendStart(Report := Report);
END_METHOD

METHOD PROTECTED _M_AppendManualInterlocks
VAR_INPUT
    TargetPath : STRING(255);
    Value : DINT;
END_VAR
VAR_IN_OUT
    Report : ST_ReleaseReport;
END_VAR
ReleaseConditions.M_AppendManual(TargetPath := TargetPath, Value := Value,
    PressRam := PressRam, Door := Door, PartSlide := PartSlide, Report := Report);
END_METHOD

METHOD PROTECTED _M_PublishStatus
SUPER^._M_PublishStatus();
OutImm.Diagnostic := Status.Diagnostic;
END_METHOD

END_FUNCTION_BLOCK

// ---- 01_PneumaticPress/Release/FB_PressDemoRelease.TcPOU
// Project-owned release engineering for the pneumatic press.
// This FB is not a Fraktal module: it exposes named condition state and fills
// the Unit's authoritative release reports without adding an OPC UA tree node.
FUNCTION_BLOCK FB_PressDemoRelease
VAR_OUTPUT
    ModeStart : FB_PermIntlk;
    ModeStartAirPressureOk : BOOL;
END_VAR
VAR
    _unitPath : STRING(255);
END_VAR

; // Evaluated explicitly by the owning Unit after child cyclic status is available.

METHOD Setup : BOOL
VAR_INPUT
    UnitPath : STRING(255);
END_VAR
_unitPath := UnitPath;
Setup := ModeStart.Define(Index := 1, Description := 'project.condition.airPressureOk',
    Reason := E_Reason.PERMISSIVE_NOT_MET, Bypassable := FALSE);
END_METHOD

METHOD M_Evaluate
VAR_INPUT
    PressRam : REFERENCE TO FB_CylinderCM;
    Door : REFERENCE TO FB_CylinderCM;
    PartSlide : REFERENCE TO FB_CylinderCM;
    TwoHand : REFERENCE TO FB_TwoHandStartCM;
    PneumaticPower : REFERENCE TO FB_PowerGroupCM;
    AirPressure : REFERENCE TO FB_AirPressureMonitorCM;
END_VAR
// Direction-specific functional collision prevention. Certified safety remains
// authoritative for hazardous-motion permission and safe output removal.
Door.SetDirectionalPermits(
    ExtendOk := PartSlide.OutImm.Extended AND NOT PartSlide.OutImm.Retracted
        AND NOT PartSlide.Busy AND NOT PartSlide.Error,
    RetractOk := TRUE,
    ExtendDescriptionKey := 'project.interlock.doorCloseRequiresSlideInside',
    RetractDescriptionKey := 'project.interlock.doorOpenPermitted');
PartSlide.SetDirectionalPermits(
    ExtendOk := Door.OutImm.Retracted AND NOT Door.OutImm.Extended
        AND NOT Door.Busy AND NOT Door.Error,
    RetractOk := Door.OutImm.Retracted AND NOT Door.OutImm.Extended
        AND NOT Door.Busy AND NOT Door.Error,
    ExtendDescriptionKey := 'project.interlock.slideMoveRequiresDoorOpen',
    RetractDescriptionKey := 'project.interlock.slideOutsideRequiresDoorOpen');
PressRam.SetDirectionalPermits(
    ExtendOk := Door.OutImm.Extended AND NOT Door.OutImm.Retracted
        AND PartSlide.OutImm.Extended AND NOT PartSlide.OutImm.Retracted
        AND NOT Door.Error AND NOT PartSlide.Error
        AND AirPressure.OutImm.PressureOk AND TwoHand.OutImm.SafeActive
        AND PneumaticPower.OutCmd.PowerOn,
    RetractOk := TRUE,
    ExtendDescriptionKey := 'project.interlock.pressRequiresGuardSlideTwoHandPower',
    RetractDescriptionKey := 'project.interlock.pressRetractPermitted');

// Mode-entry release is distinct from future AUTO waits. Part presence and the
// two-hand edge remain live conditions in the AUTO SFC action.
ModeStartAirPressureOk := AirPressure.OutImm.PressureOk;
ModeStart.Cond[1] := ModeStartAirPressureOk;
ModeStart();
END_METHOD

METHOD M_AppendStart
VAR_IN_OUT
    Report : ST_ReleaseReport;
END_VAR
ModeStart.AppendFailed(SourcePath := _unitPath, Report := Report);
END_METHOD

METHOD M_AppendManual
VAR_INPUT
    TargetPath : STRING(255);
    Value : DINT;
    PressRam : REFERENCE TO FB_CylinderCM;
    Door : REFERENCE TO FB_CylinderCM;
    PartSlide : REFERENCE TO FB_CylinderCM;
END_VAR
VAR_IN_OUT
    Report : ST_ReleaseReport;
END_VAR
IF TargetPath = PressRam.Name THEN
    PressRam.AppendDirectionalRelease(Value := Value, Report := Report);
ELSIF TargetPath = Door.Name THEN
    Door.AppendDirectionalRelease(Value := Value, Report := Report);
ELSIF TargetPath = PartSlide.Name THEN
    PartSlide.AppendDirectionalRelease(Value := Value, Report := Report);
ELSE
    IF Report.Count < PL_Fraktal.MAX_RELEASE_REASONS THEN
        Report.Count := Report.Count + 1;
        Report.Reasons[Report.Count].Description := 'std.error.unsupportedManualTarget';
        Report.Reasons[Report.Count].ReasonCode := E_Reason.UNSUPPORTED_COMMAND;
        Report.Reasons[Report.Count].SourcePath := _unitPath;
        Report.Reasons[Report.Count].Kind := E_ReleaseKind.OTHER;
        Report.Reasons[Report.Count].Bypassable := FALSE;
    ELSE
        ; // bounded report is full; no array write is attempted
    END_IF
END_IF
END_METHOD

END_FUNCTION_BLOCK

// ---- 01_PneumaticPress/Sequences/FB_PressDemoHome.TcPOU
// HOME mode chain (Core §6.2/§6.8 ST skeleton on FB_SequenceBase): establish the
// shared load-safe position, then complete. Finite (does not loop).
FUNCTION_BLOCK FB_PressDemoHome EXTENDS FB_SequenceBase
VAR
    {attribute 'OPC.UA.DA' := '0'}
    _outCmd : REFERENCE TO ST_PneumaticPressOutCmd;
    {attribute 'OPC.UA.DA' := '0'}
    _loadPosition : FB_PressDemoLoadPosition;
    _loadPositionRunning : BOOL;
END_VAR

METHOD Setup : BOOL
VAR_INPUT
    Host : I_SequenceHost;
END_VAR
VAR_IN_OUT
    PressRam : FB_CylinderCM;
    Door : FB_CylinderCM;
    PartSlide : FB_CylinderCM;
    OutCmd : ST_PneumaticPressOutCmd;
END_VAR
_outCmd REF= OutCmd;
Setup := M_Attach(Host := Host) AND __ISVALIDREF(_outCmd)
    AND _loadPosition.Setup(Host := Host, PressRam := PressRam, Door := Door, PartSlide := PartSlide);
END_METHOD

METHOD M_Reset
M_ResetBase(FirstStep := 0);
_loadPositionRunning := FALSE;
_loadPosition.M_Reset(BaseStepNo := 0);
END_METHOD

METHOD M_Run
IF NOT _attached THEN
    RETURN;
END_IF
CASE _step OF
    0:  // initialize
        M_Step(StepNo := 0, StepName := 'project.step.pressHomeInitialize',
            Awaits := 0, AwaitingLabel := '', Class := E_TimeClass.WORK, ExpectedTime := T#0S);
        _outCmd.Homed := FALSE;
        _outCmd.ChangeoverCompleted := FALSE;
        _loadPositionRunning := FALSE;
        _retVal := E_StepResult.ADVANCE;
        M_Advance(OnAdvance := 900);
    900:  // shared load-safe position (composite step, §6.7)
        IF NOT _loadPositionRunning THEN
            _loadPosition.M_Reset(BaseStepNo := 900);
            _loadPositionRunning := TRUE;
        END_IF
        _loadPosition.M_Run();
        IF _loadPosition.Done THEN
            _loadPositionRunning := FALSE;
            _retVal := E_StepResult.ADVANCE;
        END_IF
        M_Advance(OnAdvance := 999);
    999:  // complete
        M_Step(StepNo := 999, StepName := 'project.step.pressHomeComplete',
            Awaits := 0, AwaitingLabel := '', Class := E_TimeClass.WORK, ExpectedTime := T#0S);
        _outCmd.Homed := TRUE;
        M_Complete();
ELSE
    M_Fault(Reason := E_Reason.STEP_STALLED, DescriptionKey := 'std.error.undefinedStep');
END_CASE
END_METHOD

END_FUNCTION_BLOCK

// ---- 01_PneumaticPress/Sequences/FB_PressDemoLoadPosition.TcPOU
// Shared load-safe-position sub-sequence (Core §6.7): ram up, door open, slide
// outside. HOME and CHANGEOVER both embed it as one composite step, passing a
// BaseStepNo window so its detailed progress projects through the Unit's normal
// §6.5 step record. Implemented as a Core §6.8 ST `CASE _step OF` skeleton on
// FB_SequenceBase — the step actions issue child commands only through the §6.1
// handshake (M_MayIssue), and progression rides the shared _retVal via M_Advance.
FUNCTION_BLOCK FB_PressDemoLoadPosition EXTENDS FB_SequenceBase
VAR
    _baseStepNo : INT;
    {attribute 'OPC.UA.DA' := '0'}
    _pressRam : REFERENCE TO FB_CylinderCM;
    {attribute 'OPC.UA.DA' := '0'}
    _door : REFERENCE TO FB_CylinderCM;
    {attribute 'OPC.UA.DA' := '0'}
    _partSlide : REFERENCE TO FB_CylinderCM;
END_VAR

// step body runs via M_Run; the Unit calls this instance each scan

METHOD Setup : BOOL
VAR_INPUT
    Host : I_SequenceHost;
END_VAR
VAR_IN_OUT
    PressRam : FB_CylinderCM;
    Door : FB_CylinderCM;
    PartSlide : FB_CylinderCM;
END_VAR
_pressRam REF= PressRam;
_door REF= Door;
_partSlide REF= PartSlide;
Setup := M_Attach(Host := Host)
    AND __ISVALIDREF(_pressRam) AND __ISVALIDREF(_door) AND __ISVALIDREF(_partSlide);
END_METHOD

METHOD M_Reset
VAR_INPUT
    BaseStepNo : INT;
END_VAR
_baseStepNo := BaseStepNo;
M_ResetBase(FirstStep := 0);
END_METHOD

// §6.8 ST step skeleton. One M_Step per step, one commit via M_Advance.
METHOD M_Run
IF NOT _attached THEN
    RETURN;
END_IF
CASE _step OF
    0:  // ram up
        M_Step(StepNo := _baseStepNo, StepName := 'project.step.pressSafePositionRamUp',
            Awaits := _pressRam, AwaitingLabel := 'PressRam.RETRACT',
            Class := E_TimeClass.WORK, ExpectedTime := T#0S);
        IF M_MayIssue(Steppable := TRUE) THEN
            _pressRam.Abort := FALSE;
            _pressRam.Command := E_CylinderCommand.RETRACT;
            _pressRam.Execute := TRUE;
        END_IF
        IF _pressRam.Done THEN
            _pressRam.Execute := FALSE;
            _retVal := E_StepResult.ADVANCE;
        END_IF
        M_Advance(OnAdvance := 20);
    20:  // door open
        M_Step(StepNo := _baseStepNo + 20, StepName := 'project.step.pressSafePositionDoorOpen',
            Awaits := _door, AwaitingLabel := 'Door.RETRACT',
            Class := E_TimeClass.WORK, ExpectedTime := T#0S);
        IF M_MayIssue(Steppable := TRUE) THEN
            _door.Abort := FALSE;
            _door.Command := E_CylinderCommand.RETRACT;
            _door.Execute := TRUE;
        END_IF
        IF _door.Done THEN
            _door.Execute := FALSE;
            _retVal := E_StepResult.ADVANCE;
        END_IF
        M_Advance(OnAdvance := 40);
    40:  // slide outside
        M_Step(StepNo := _baseStepNo + 40, StepName := 'project.step.pressSafePositionSlideOutside',
            Awaits := _partSlide, AwaitingLabel := 'PartSlide.RETRACT',
            Class := E_TimeClass.WORK, ExpectedTime := T#0S);
        IF M_MayIssue(Steppable := TRUE) THEN
            _partSlide.Abort := FALSE;
            _partSlide.Command := E_CylinderCommand.RETRACT;
            _partSlide.Execute := TRUE;
        END_IF
        IF _partSlide.Done THEN
            _partSlide.Execute := FALSE;
            _retVal := E_StepResult.ADVANCE;
        END_IF
        M_Advance(OnAdvance := 999);
    999:  // established
        M_Step(StepNo := _baseStepNo + 60, StepName := 'project.step.pressSafePositionComplete',
            Awaits := 0, AwaitingLabel := '', Class := E_TimeClass.WORK, ExpectedTime := T#0S);
        Done := TRUE;
ELSE
    M_Fault(Reason := E_Reason.STEP_STALLED, DescriptionKey := 'std.error.undefinedStep');
END_CASE
END_METHOD

END_FUNCTION_BLOCK

// ---- 01_PneumaticPress/Sequences/FB_PressDemoChangeover.TcPOU
// CHANGEOVER mode chain (Core §6.2/§6.8 ST skeleton on FB_SequenceBase): validate
// the selected model, establish the shared load-safe position, then ask the
// operator (§6.11) to confirm tooling/material match before completing. The
// 'repeat position' answer restarts the guided move via a backward jump (§6.10).
FUNCTION_BLOCK FB_PressDemoChangeover EXTENDS FB_SequenceBase
VAR
    _decisionRequest : ST_DecisionRequest;
    _answer : INT;
    _modelSelected : BOOL;
    {attribute 'OPC.UA.DA' := '0'}
    _outCmd : REFERENCE TO ST_PneumaticPressOutCmd;
    {attribute 'OPC.UA.DA' := '0'}
    _model : REFERENCE TO ST_ModelId;
    {attribute 'OPC.UA.DA' := '0'}
    _loadPosition : FB_PressDemoLoadPosition;
    _loadPositionRunning : BOOL;
END_VAR

METHOD Setup : BOOL
VAR_INPUT
    Host : I_SequenceHost;
END_VAR
VAR_IN_OUT
    PressRam : FB_CylinderCM;
    Door : FB_CylinderCM;
    PartSlide : FB_CylinderCM;
    OutCmd : ST_PneumaticPressOutCmd;
    Model : ST_ModelId;
END_VAR
_outCmd REF= OutCmd;
_model REF= Model;
Setup := M_Attach(Host := Host) AND __ISVALIDREF(_outCmd) AND __ISVALIDREF(_model)
    AND _loadPosition.Setup(Host := Host, PressRam := PressRam, Door := Door, PartSlide := PartSlide);
END_METHOD

METHOD M_Reset
M_ResetBase(FirstStep := 0);
_answer := 0;
_loadPositionRunning := FALSE;
_loadPosition.M_Reset(BaseStepNo := 0);
END_METHOD

METHOD M_Run
IF NOT _attached THEN
    RETURN;
END_IF
CASE _step OF
    0:  // initialize
        M_Step(StepNo := 0, StepName := 'project.step.pressChangeoverInitialize',
            Awaits := 0, AwaitingLabel := '', Class := E_TimeClass.WORK, ExpectedTime := T#0S);
        _outCmd.ChangeoverCompleted := FALSE;
        _outCmd.Homed := FALSE;
        _answer := 0;
        _decisionRequest.Prompt := '';
        M_ClearDecision();
        _loadPositionRunning := FALSE;
        _retVal := E_StepResult.ADVANCE;
        M_Advance(OnAdvance := 800);
    800:  // validate the transactionally-loaded model
        M_Step(StepNo := 800, StepName := 'project.step.pressChangeoverValidateModel',
            Awaits := 0, AwaitingLabel := '', Class := E_TimeClass.WAIT_OPERATOR, ExpectedTime := T#0S);
        _modelSelected := M_Await(Idx := 1, Label := 'project.condition.pressModelSelected',
            Ok := _model.ModelCode <> '');
        IF _modelSelected THEN
            _loadPositionRunning := FALSE;
            _retVal := E_StepResult.ADVANCE;
        END_IF
        M_Advance(OnAdvance := 810);
    810:  // shared load-safe position (composite step)
        IF NOT _loadPositionRunning THEN
            _loadPosition.M_Reset(BaseStepNo := 810);
            _loadPositionRunning := TRUE;
        END_IF
        _loadPosition.M_Run();
        IF _loadPosition.Done THEN
            _loadPositionRunning := FALSE;
            _retVal := E_StepResult.ADVANCE;
        END_IF
        M_Advance(OnAdvance := 870);
    870:  // request tooling/material confirmation
        M_Step(StepNo := 870, StepName := 'project.step.pressChangeoverRequestConfirmation',
            Awaits := 0, AwaitingLabel := '', Class := E_TimeClass.WAIT_OPERATOR, ExpectedTime := T#0S);
        _decisionRequest.Prompt := 'project.decision.pressChangeoverConfirm';
        _decisionRequest.Options[1] := 'project.decision.confirmChangeover';
        _decisionRequest.Options[2] := 'project.decision.repeatChangeoverPosition';
        _decisionRequest.Default := 0;
        _decisionRequest.Timeout := T#0S;
        M_AskDecision(Req := _decisionRequest);
        _retVal := E_StepResult.ADVANCE;
        M_Advance(OnAdvance := 880);
    880:  // await confirmation; JUMP1 = repeat the guided position
        M_Step(StepNo := 880, StepName := 'project.step.pressChangeoverAwaitConfirmation',
            Awaits := 0, AwaitingLabel := '', Class := E_TimeClass.WAIT_OPERATOR, ExpectedTime := T#0S);
        _answer := M_TakeDecision();
        IF _answer = 1 THEN
            _retVal := E_StepResult.ADVANCE;
        ELSIF _answer = 2 THEN
            _loadPositionRunning := FALSE;      // repeat the guided position from the start
            _retVal := E_StepResult.JUMP1;
        ELSE
            _modelSelected := M_Await(Idx := 1,
                Label := 'project.condition.pressChangeoverConfirmation', Ok := FALSE);
        END_IF
        M_Advance(OnAdvance := 999, OnJump1 := 810);
    999:  // complete
        M_Step(StepNo := 999, StepName := 'project.step.pressChangeoverComplete',
            Awaits := 0, AwaitingLabel := '', Class := E_TimeClass.WORK, ExpectedTime := T#0S);
        _outCmd.Homed := TRUE;
        _outCmd.ChangeoverCompleted := TRUE;
        M_Complete();
ELSE
    M_Fault(Reason := E_Reason.STEP_STALLED, DescriptionKey := 'std.error.undefinedStep');
END_CASE
END_METHOD

END_FUNCTION_BLOCK

// ---- 01_PneumaticPress/Sequences/FB_PressDemoAuto.TcPOU
// AUTO mode chain (Core §6.2/§6.8 ST skeleton on FB_SequenceBase): the continuous
// production cycle — await a fresh two-hand start with part+air present, transfer
// the part in, press for the recipe dwell, return to load position, count the good
// part, and loop until Stop. A Stop requested at the between-cycles wait is honored
// there (M_StopNow) so no phantom cycle is charged. Every child motion goes through
// the §6.1 handshake (M_MayIssue); progression rides the shared _retVal.
FUNCTION_BLOCK FB_PressDemoAuto EXTENDS FB_SequenceBase
VAR
    _settle : TON;
    _partReady, _airReady, _startReady : BOOL;
    _traceAccepted, _recordAccepted, _partProcessed : BOOL;
    {attribute 'OPC.UA.DA' := '0'}
    _pressRam : REFERENCE TO FB_CylinderCM;
    {attribute 'OPC.UA.DA' := '0'}
    _door : REFERENCE TO FB_CylinderCM;
    {attribute 'OPC.UA.DA' := '0'}
    _partSlide : REFERENCE TO FB_CylinderCM;
    {attribute 'OPC.UA.DA' := '0'}
    _twoHand : REFERENCE TO FB_TwoHandStartCM;
    {attribute 'OPC.UA.DA' := '0'}
    _partPresentSensor : REFERENCE TO FB_DigitalInputCM;
    {attribute 'OPC.UA.DA' := '0'}
    _airPressureMonitor : REFERENCE TO FB_AirPressureMonitorCM;
    {attribute 'OPC.UA.DA' := '0'}
    _parCfg : REFERENCE TO ST_PneumaticPressParCfg;
    {attribute 'OPC.UA.DA' := '0'}
    _outCmd : REFERENCE TO ST_PneumaticPressOutCmd;
    {attribute 'OPC.UA.DA' := '0'}
    _startLatched : REFERENCE TO BOOL;
    {attribute 'OPC.UA.DA' := '0'}
    _loadPosition : FB_PressDemoLoadPosition;
    _loadPositionRunning : BOOL;
END_VAR

METHOD Setup : BOOL
VAR_INPUT
    Host : I_SequenceHost;
END_VAR
VAR_IN_OUT
    PressRam : FB_CylinderCM;
    Door : FB_CylinderCM;
    PartSlide : FB_CylinderCM;
    TwoHand : FB_TwoHandStartCM;
    PartPresentSensor : FB_DigitalInputCM;
    AirPressureMonitor : FB_AirPressureMonitorCM;
    ParCfg : ST_PneumaticPressParCfg;
    OutCmd : ST_PneumaticPressOutCmd;
    StartLatched : BOOL;
END_VAR
_pressRam REF= PressRam;
_door REF= Door;
_partSlide REF= PartSlide;
_twoHand REF= TwoHand;
_partPresentSensor REF= PartPresentSensor;
_airPressureMonitor REF= AirPressureMonitor;
_parCfg REF= ParCfg;
_outCmd REF= OutCmd;
_startLatched REF= StartLatched;
Setup := M_Attach(Host := Host) AND __ISVALIDREF(_pressRam) AND __ISVALIDREF(_door)
    AND __ISVALIDREF(_partSlide) AND __ISVALIDREF(_twoHand)
    AND __ISVALIDREF(_partPresentSensor) AND __ISVALIDREF(_airPressureMonitor)
    AND __ISVALIDREF(_parCfg) AND __ISVALIDREF(_outCmd) AND __ISVALIDREF(_startLatched)
    AND _loadPosition.Setup(Host := Host, PressRam := PressRam, Door := Door, PartSlide := PartSlide);
END_METHOD

METHOD M_Reset
M_ResetBase(FirstStep := 0);
_settle(IN := FALSE);
_loadPositionRunning := FALSE;
_loadPosition.M_Reset(BaseStepNo := 0);
END_METHOD

METHOD M_Run
IF NOT _attached THEN
    RETURN;
END_IF
CASE _step OF
    0:  // initialize
        M_Step(StepNo := 0, StepName := 'project.step.pressAutoInitialize',
            Awaits := 0, AwaitingLabel := '', Class := E_TimeClass.WORK, ExpectedTime := T#0S);
        _outCmd.CycleCompleted := FALSE;
        _outCmd.Homed := FALSE;
        _outCmd.ChangeoverCompleted := FALSE;
        _loadPositionRunning := FALSE;
        _retVal := E_StepResult.ADVANCE;
        M_Advance(OnAdvance := 100);
    100:  // await a fresh two-hand start (the §8.11.1 cycle-start marker)
        M_Step(StepNo := 100, StepName := 'project.step.pressAwaitTwoHand',
            Awaits := 0, AwaitingLabel := '', Class := E_TimeClass.WAIT_OPERATOR, ExpectedTime := T#0S);
        _outCmd.CycleCompleted := FALSE;
        _partReady := M_Await(Idx := 1, Label := 'project.condition.partPresent',
            Ok := _partPresentSensor.OutImm.Value AND _partPresentSensor.OutImm.Quality);
        _airReady := M_Await(Idx := 2, Label := 'project.condition.airPressureOk',
            Ok := _airPressureMonitor.OutImm.PressureOk);
        IF _parCfg.RequireTwoHandStart THEN
            _startReady := M_Await(Idx := 3, Label := 'project.condition.twoHandStart', Ok := _startLatched);
        ELSE
            _startReady := TRUE;
        END_IF
        IF M_StopPending() THEN
            M_StopNow();                       // stop accepted BETWEEN cycles: no phantom cycle
        ELSIF _partReady AND _airReady AND _startReady THEN
            _traceAccepted := M_PartReceived();
            _retVal := E_StepResult.ADVANCE;
        END_IF
        M_Advance(OnAdvance := 110);
    110:  // ram up
        M_Step(StepNo := 110, StepName := 'project.step.pressRamUp',
            Awaits := _pressRam, AwaitingLabel := 'PressRam.RETRACT', Class := E_TimeClass.WORK, ExpectedTime := T#0S);
        IF M_MayIssue(Steppable := TRUE) THEN
            _pressRam.Abort := FALSE; _pressRam.Command := E_CylinderCommand.RETRACT; _pressRam.Execute := TRUE;
        END_IF
        IF _pressRam.Done THEN _pressRam.Execute := FALSE; _retVal := E_StepResult.ADVANCE; END_IF
        M_Advance(OnAdvance := 130);
    130:  // door open
        M_Step(StepNo := 130, StepName := 'project.step.pressDoorOpen',
            Awaits := _door, AwaitingLabel := 'Door.RETRACT', Class := E_TimeClass.WORK, ExpectedTime := T#0S);
        IF M_MayIssue(Steppable := TRUE) THEN
            _door.Abort := FALSE; _door.Command := E_CylinderCommand.RETRACT; _door.Execute := TRUE;
        END_IF
        IF _door.Done THEN _door.Execute := FALSE; _retVal := E_StepResult.ADVANCE; END_IF
        M_Advance(OnAdvance := 150);
    150:  // slide inside (value-adding sequence begins)
        M_Step(StepNo := 150, StepName := 'project.step.pressSlideInside',
            Awaits := _partSlide, AwaitingLabel := 'PartSlide.EXTEND', Class := E_TimeClass.WORK, ExpectedTime := T#0S);
        IF M_MayIssue(Steppable := TRUE) THEN
            M_PartStarted();
            _partSlide.Abort := FALSE; _partSlide.Command := E_CylinderCommand.EXTEND; _partSlide.Execute := TRUE;
        END_IF
        IF _partSlide.Done THEN _partSlide.Execute := FALSE; _retVal := E_StepResult.ADVANCE; END_IF
        M_Advance(OnAdvance := 170);
    170:  // transfer settle
        M_Step(StepNo := 170, StepName := 'project.step.pressTransferSettle',
            Awaits := 0, AwaitingLabel := '', Class := E_TimeClass.WORK, ExpectedTime := _parCfg.TransferSettleTime);
        _retVal := M_Delay(PT := _parCfg.TransferSettleTime);
        M_Advance(OnAdvance := 180);
    180:  // door close
        M_Step(StepNo := 180, StepName := 'project.step.pressDoorClose',
            Awaits := _door, AwaitingLabel := 'Door.EXTEND', Class := E_TimeClass.WORK, ExpectedTime := T#0S);
        IF M_MayIssue(Steppable := TRUE) THEN
            _door.Abort := FALSE; _door.Command := E_CylinderCommand.EXTEND; _door.Execute := TRUE;
        END_IF
        IF _door.Done THEN _door.Execute := FALSE; _retVal := E_StepResult.ADVANCE; END_IF
        M_Advance(OnAdvance := 200);
    200:  // ram down
        M_Step(StepNo := 200, StepName := 'project.step.pressRamDown',
            Awaits := _pressRam, AwaitingLabel := 'PressRam.EXTEND', Class := E_TimeClass.WORK, ExpectedTime := T#0S);
        IF M_MayIssue(Steppable := TRUE) THEN
            _pressRam.Abort := FALSE; _pressRam.Command := E_CylinderCommand.EXTEND; _pressRam.Execute := TRUE;
        END_IF
        IF _pressRam.Done THEN _pressRam.Execute := FALSE; _retVal := E_StepResult.ADVANCE; END_IF
        M_Advance(OnAdvance := 220);
    220:  // press dwell — two-hand must stay active
        M_Step(StepNo := 220, StepName := 'project.step.pressDwell',
            Awaits := 0, AwaitingLabel := '', Class := E_TimeClass.WORK, ExpectedTime := _parCfg.PressSettleTime);
        IF NOT _twoHand.OutImm.SafeActive AND _parCfg.RequireTwoHandStart THEN
            _pressRam.WithdrawOutputs();
            M_Fault(Reason := E_Reason.INTERLOCK_DROPPED, DescriptionKey := 'project.error.twoHandReleasedDuringPress');
        ELSE
            _retVal := M_Delay(PT := _parCfg.PressSettleTime);
        END_IF
        M_Advance(OnAdvance := 230);
    230:  // record the applied dwell (§3.16.1 measured value)
        M_Step(StepNo := 230, StepName := 'project.step.pressRecordResult',
            Awaits := 0, AwaitingLabel := '', Class := E_TimeClass.WORK, ExpectedTime := T#0S);
        _recordAccepted := M_PartRecord(RecordName := 'PressDwell',
            Value := DINT_TO_LREAL(TIME_TO_DINT(_parCfg.PressSettleTime)),
            Minimum := 0, Maximum := 30000,
            Target := DINT_TO_LREAL(TIME_TO_DINT(_parCfg.PressSettleTime)), EngUnit := 'ms');
        _loadPositionRunning := FALSE;
        _retVal := E_StepResult.ADVANCE;
        M_Advance(OnAdvance := 240);
    240:  // return to the shared load-safe position (composite step)
        IF NOT _loadPositionRunning THEN
            _loadPosition.M_Reset(BaseStepNo := 240);
            _loadPositionRunning := TRUE;
        END_IF
        _loadPosition.M_Run();
        IF _loadPosition.Done THEN
            _loadPositionRunning := FALSE;
            _retVal := E_StepResult.ADVANCE;
        END_IF
        M_Advance(OnAdvance := 999);
    999:  // cycle complete — write result, count by verdict, loop (§8.11.1 finish marker)
        M_Step(StepNo := 999, StepName := 'project.step.pressAutoComplete',
            Awaits := 0, AwaitingLabel := '', Class := E_TimeClass.WORK, ExpectedTime := T#0S);
        _outCmd.CycleCompleted := TRUE;
        _partProcessed := M_PartProcessed(Verdict := E_Verdict.OK, Reason := E_Reason.NONE);
        IF NOT _partProcessed THEN
            M_CountGood();                     // §3.9: no carrier configured — count directly
        END_IF
        _startLatched := FALSE;
        IF M_EndOfCycle() THEN
            _retVal := E_StepResult.ADVANCE;   // stop NOT requested: loop to N100
        END_IF
        M_Advance(OnAdvance := 100);
ELSE
    M_Fault(Reason := E_Reason.STEP_STALLED, DescriptionKey := 'std.error.undefinedStep');
END_CASE
END_METHOD

END_FUNCTION_BLOCK

// ---- 01_PneumaticPress/Io/FB_PressIoCatalog.TcPOU
// Owner-local I/O engineering-data adapter. This is the ONE source for the approved
// tag/address/description/module-role join. It contains no cyclic behavior,
// process-image access, topology algorithms or device logic.
FUNCTION_BLOCK FB_PressIoCatalog
VAR
    _publisher : FB_IoTopologyPublisher;
    _rootPath : STRING(255);
END_VAR

;

METHOD Setup : BOOL
VAR_INPUT
    UnitRef : REFERENCE TO FB_PressDemoUnit;
END_VAR
VAR
    Ok : BOOL;
    SlideIdentity, DoorIdentity, PressIdentity : ST_CylinderIoIdentity;
    PartIdentity, LowAirIdentity, OperatingAirIdentity : ST_IoPointIdentity;
END_VAR
_rootPath := UnitRef.Name;
Ok := _publisher.Setup(DataRef := GVL_PressFieldbus.Topology, ResetData := TRUE);
Ok := _publisher.M_DefineNode(Index := 1, Name := '=000+S-A610-A1',
    DescriptionKey := 'project.hardware.cx2030', TypeId := 'Beckhoff CX2030',
    Address := 'EtherCAT master', ParentIndex := 0) AND Ok;
Ok := _publisher.M_DefineNode(Index := 2, Name := '=000+S-K010',
    DescriptionKey := 'project.hardware.ek1200', TypeId := 'Beckhoff EK1200-5000',
    Address := 'EtherCAT Box 1', ParentIndex := 1) AND Ok;
Ok := _publisher.M_DefineNode(Index := 3, Name := '=000+S-K010B1',
    DescriptionKey := 'project.hardware.el1809', TypeId := 'Beckhoff EL1809',
    Address := 'EtherCAT Box 2', ParentIndex := 2) AND Ok;
Ok := _publisher.M_DefineNode(Index := 4, Name := '=000+S-K010C1',
    DescriptionKey := 'project.hardware.el2809', TypeId := 'Beckhoff EL2809',
    Address := 'EtherCAT Box 3', ParentIndex := 2) AND Ok;
Ok := _publisher.M_DefineNode(Index := 5, Name := '=000+S-K010D1',
    DescriptionKey := 'project.hardware.el6001', TypeId := 'Beckhoff EL6001 RS232',
    Address := 'EtherCAT Box 4', ParentIndex := 2) AND Ok;
Ok := _publisher.M_DefineNode(Index := 6, Name := '=000+S-K010E',
    DescriptionKey := 'project.hardware.el9011', TypeId := 'Beckhoff EL9011',
    Address := 'EtherCAT Box 5', ParentIndex := 2) AND Ok;

Ok := _M_DefineCylinder(Identity := SlideIdentity,
    ModulePath := UnitRef.PartSlide.Name,
    ExtendedSensorTag := '_101B301A', ExtendedSensorDescription := 'project.io.101B301A',
    ExtendedSensorAddress := '=000+S-K010B1 Ch1', ExtendedSensorIndex := 1,
    RetractedSensorTag := '_101B301B', RetractedSensorDescription := 'project.io.101B301B',
    RetractedSensorAddress := '=000+S-K010B1 Ch2', RetractedSensorIndex := 2,
    ExtendOutputTag := '_101K301A', ExtendOutputDescription := 'project.io.101K301A',
    ExtendOutputAddress := '=000+S-K010C1 Ch1', ExtendOutputIndex := 1,
    RetractOutputTag := '_101K301B', RetractOutputDescription := 'project.io.101K301B',
    RetractOutputAddress := '=000+S-K010C1 Ch2', RetractOutputIndex := 2,
    ExtendedTimeoutKey := 'project.error.slideInsideSensorTimeout',
    RetractedTimeoutKey := 'project.error.slideOutsideSensorTimeout',
    BothSensorsKey := 'project.error.slidePositionSensorsConflict') AND Ok;
UnitRef.PartSlide.ConfigureIoIdentity(Identity := SlideIdentity);
Ok := _M_DefineCylinder(Identity := DoorIdentity,
    ModulePath := UnitRef.Door.Name,
    ExtendedSensorTag := '_101B201A', ExtendedSensorDescription := 'project.io.101B201A',
    ExtendedSensorAddress := '=000+S-K010B1 Ch3', ExtendedSensorIndex := 3,
    RetractedSensorTag := '_101B201B', RetractedSensorDescription := 'project.io.101B201B',
    RetractedSensorAddress := '=000+S-K010B1 Ch4', RetractedSensorIndex := 4,
    ExtendOutputTag := '_101K201A', ExtendOutputDescription := 'project.io.101K201A',
    ExtendOutputAddress := '=000+S-K010C1 Ch3', ExtendOutputIndex := 3,
    RetractOutputTag := '_101K201B', RetractOutputDescription := 'project.io.101K201B',
    RetractOutputAddress := '=000+S-K010C1 Ch4', RetractOutputIndex := 4,
    ExtendedTimeoutKey := 'project.error.doorClosedSensorTimeout',
    RetractedTimeoutKey := 'project.error.doorOpenSensorTimeout',
    BothSensorsKey := 'project.error.doorPositionSensorsConflict') AND Ok;
UnitRef.Door.ConfigureIoIdentity(Identity := DoorIdentity);
Ok := _M_DefineCylinder(Identity := PressIdentity,
    ModulePath := UnitRef.PressRam.Name,
    ExtendedSensorTag := '_101B202A', ExtendedSensorDescription := 'project.io.101B202A',
    ExtendedSensorAddress := '=000+S-K010B1 Ch5', ExtendedSensorIndex := 5,
    RetractedSensorTag := '_101B202B', RetractedSensorDescription := 'project.io.101B202B',
    RetractedSensorAddress := '=000+S-K010B1 Ch6', RetractedSensorIndex := 6,
    ExtendOutputTag := '_101K202A', ExtendOutputDescription := 'project.io.101K202A',
    ExtendOutputAddress := '=000+S-K010C1 Ch5', ExtendOutputIndex := 5,
    RetractOutputTag := '_101K202B', RetractOutputDescription := 'project.io.101K202B',
    RetractOutputAddress := '=000+S-K010C1 Ch6', RetractOutputIndex := 6,
    ExtendedTimeoutKey := 'project.error.pressDownSensorTimeout',
    RetractedTimeoutKey := 'project.error.pressUpSensorTimeout',
    BothSensorsKey := 'project.error.pressPositionSensorsConflict') AND Ok;
UnitRef.PressRam.ConfigureIoIdentity(Identity := PressIdentity);

Ok := _M_DefinePoint(NodeIndex := 3, ChannelIndex := 7, Tag := '_101S101',
    DescriptionKey := 'project.io.101S101', Address := '=000+S-K010B1 Ch7',
    ModulePath := UnitRef.TwoHand.Name, Dir := E_ChannelDir.INPUT) AND Ok;
Ok := _M_DefinePoint(NodeIndex := 3, ChannelIndex := 8, Tag := '_101S102',
    DescriptionKey := 'project.io.101S102', Address := '=000+S-K010B1 Ch8',
    ModulePath := UnitRef.TwoHand.Name, Dir := E_ChannelDir.INPUT) AND Ok;
LowAirIdentity.Tag := '_000MB085A_2';
LowAirIdentity.DescriptionKey := 'project.io.000MB085A_2';
LowAirIdentity.Address := '=000+S-K010B1 Ch10';
LowAirIdentity.ModulePath := UnitRef.AirPressureMonitor.Name;
LowAirIdentity.Path := CONCAT(_rootPath, '.IO._000MB085A_2');
Ok := _M_DefineIdentity(NodeIndex := 3, ChannelIndex := 9,
    Identity := LowAirIdentity, Dir := E_ChannelDir.INPUT) AND Ok;
OperatingAirIdentity.Tag := '_000MB085A_4';
OperatingAirIdentity.DescriptionKey := 'project.io.000MB085A_4';
OperatingAirIdentity.Address := '=000+S-K010B1 Ch11';
OperatingAirIdentity.ModulePath := UnitRef.AirPressureMonitor.Name;
OperatingAirIdentity.Path := CONCAT(_rootPath, '.IO._000MB085A_4');
Ok := _M_DefineIdentity(NodeIndex := 3, ChannelIndex := 10,
    Identity := OperatingAirIdentity, Dir := E_ChannelDir.INPUT) AND Ok;
UnitRef.AirPressureMonitor.ConfigureIoIdentity(LowSensor := LowAirIdentity,
    OperatingSensor := OperatingAirIdentity);
PartIdentity.Tag := '_101B601';
PartIdentity.DescriptionKey := 'project.io.101B601';
PartIdentity.Address := '=000+S-K010B1 Ch12';
PartIdentity.ModulePath := UnitRef.PartPresentSensor.Name;
PartIdentity.Path := CONCAT(_rootPath, '.IO._101B601');
Ok := _M_DefineIdentity(NodeIndex := 3, ChannelIndex := 11,
    Identity := PartIdentity, Dir := E_ChannelDir.INPUT) AND Ok;
UnitRef.PartPresentSensor.ConfigureIoIdentity(Identity := PartIdentity);
Ok := _M_DefinePoint(NodeIndex := 3, ChannelIndex := 12, Tag := '_000K911_Y32',
    DescriptionKey := 'project.io.000K911_Y32', Address := '=000+S-K010B1 Ch14',
    ModulePath := UnitRef.PneumaticPower.Name, Dir := E_ChannelDir.INPUT) AND Ok;
Ok := _M_DefinePoint(NodeIndex := 3, ChannelIndex := 13, Tag := '_000K910A',
    DescriptionKey := 'project.io.000K910A', Address := '=000+S-K010B1 Ch15',
    ModulePath := UnitRef.Name, Dir := E_ChannelDir.INPUT) AND Ok;
Ok := _M_DefinePoint(NodeIndex := 4, ChannelIndex := 7, Tag := '_101P101',
    DescriptionKey := 'project.io.101P101', Address := '=000+S-K010C1 Ch7',
    ModulePath := UnitRef.TwoHand.Name, Dir := E_ChannelDir.OUTPUT) AND Ok;
Ok := _M_DefinePoint(NodeIndex := 4, ChannelIndex := 8, Tag := '_101P102',
    DescriptionKey := 'project.io.101P102', Address := '=000+S-K010C1 Ch8',
    ModulePath := UnitRef.TwoHand.Name, Dir := E_ChannelDir.OUTPUT) AND Ok;
Ok := _M_DefinePoint(NodeIndex := 4, ChannelIndex := 9, Tag := '_000K951_A1',
    DescriptionKey := 'project.io.000K951_A1', Address := '=000+S-K010C1 Ch10',
    ModulePath := UnitRef.PneumaticPower.Name, Dir := E_ChannelDir.OUTPUT) AND Ok;
Ok := _M_DefinePoint(NodeIndex := 4, ChannelIndex := 10, Tag := '_000K911_A1',
    DescriptionKey := 'project.io.000K911_A1', Address := '=000+S-K010C1 Ch11',
    ModulePath := UnitRef.PneumaticPower.Name, Dir := E_ChannelDir.OUTPUT) AND Ok;
Setup := _publisher.M_Validate() AND Ok;
END_METHOD

METHOD PRIVATE _M_DefineIdentity : BOOL
VAR_INPUT
    NodeIndex : INT;
    ChannelIndex : INT;
    Identity : ST_IoPointIdentity;
    Dir : E_ChannelDir;
END_VAR
_M_DefineIdentity := _publisher.M_DefineDigitalChannel(
    NodeIndex := NodeIndex, ChannelIndex := ChannelIndex, Tag := Identity.Tag,
    DescriptionKey := Identity.DescriptionKey, Address := Identity.Address,
    Path := Identity.Path, ModulePath := Identity.ModulePath, Dir := Dir);
END_METHOD

METHOD PRIVATE _M_DefinePoint : BOOL
VAR_INPUT
    NodeIndex : INT;
    ChannelIndex : INT;
    Tag : STRING(80);
    DescriptionKey : STRING(160);
    Address : STRING(80);
    ModulePath : STRING(255);
    Dir : E_ChannelDir;
END_VAR
VAR
    Path : STRING(255);
END_VAR
Path := CONCAT(_rootPath, CONCAT('.IO.', Tag));
_M_DefinePoint := _publisher.M_DefineDigitalChannel(NodeIndex := NodeIndex,
    ChannelIndex := ChannelIndex, Tag := Tag, DescriptionKey := DescriptionKey,
    Address := Address, Path := Path, ModulePath := ModulePath, Dir := Dir);
END_METHOD

METHOD PRIVATE _M_DefineCylinder : BOOL
VAR_INPUT
    ModulePath : STRING(255);
    ExtendedSensorTag : STRING(80);
    ExtendedSensorDescription : STRING(160);
    ExtendedSensorAddress : STRING(80);
    ExtendedSensorIndex : INT;
    RetractedSensorTag : STRING(80);
    RetractedSensorDescription : STRING(160);
    RetractedSensorAddress : STRING(80);
    RetractedSensorIndex : INT;
    ExtendOutputTag : STRING(80);
    ExtendOutputDescription : STRING(160);
    ExtendOutputAddress : STRING(80);
    ExtendOutputIndex : INT;
    RetractOutputTag : STRING(80);
    RetractOutputDescription : STRING(160);
    RetractOutputAddress : STRING(80);
    RetractOutputIndex : INT;
    ExtendedTimeoutKey : STRING(255);
    RetractedTimeoutKey : STRING(255);
    BothSensorsKey : STRING(255);
END_VAR
VAR_IN_OUT
    Identity : ST_CylinderIoIdentity;
END_VAR
VAR
    Ok : BOOL;
END_VAR
Identity.ExtendedSensor.Tag := ExtendedSensorTag;
Identity.ExtendedSensor.Address := ExtendedSensorAddress;
Identity.ExtendedSensor.DescriptionKey := ExtendedSensorDescription;
Identity.ExtendedSensor.ModulePath := ModulePath;
Identity.ExtendedSensor.Path := CONCAT(_rootPath, CONCAT('.IO.', ExtendedSensorTag));
Identity.RetractedSensor.Tag := RetractedSensorTag;
Identity.RetractedSensor.Address := RetractedSensorAddress;
Identity.RetractedSensor.DescriptionKey := RetractedSensorDescription;
Identity.RetractedSensor.ModulePath := ModulePath;
Identity.RetractedSensor.Path := CONCAT(_rootPath, CONCAT('.IO.', RetractedSensorTag));
Identity.ExtendOutput.Tag := ExtendOutputTag;
Identity.ExtendOutput.Address := ExtendOutputAddress;
Identity.ExtendOutput.DescriptionKey := ExtendOutputDescription;
Identity.ExtendOutput.ModulePath := ModulePath;
Identity.ExtendOutput.Path := CONCAT(_rootPath, CONCAT('.IO.', ExtendOutputTag));
Identity.RetractOutput.Tag := RetractOutputTag;
Identity.RetractOutput.Address := RetractOutputAddress;
Identity.RetractOutput.DescriptionKey := RetractOutputDescription;
Identity.RetractOutput.ModulePath := ModulePath;
Identity.RetractOutput.Path := CONCAT(_rootPath, CONCAT('.IO.', RetractOutputTag));
Identity.ExtendedTimeoutKey := ExtendedTimeoutKey;
Identity.RetractedTimeoutKey := RetractedTimeoutKey;
Identity.BothSensorsKey := BothSensorsKey;
Ok := _publisher.M_DefineDigitalChannel(NodeIndex := 3, ChannelIndex := ExtendedSensorIndex,
    Tag := Identity.ExtendedSensor.Tag, DescriptionKey := Identity.ExtendedSensor.DescriptionKey,
    Address := Identity.ExtendedSensor.Address, Path := Identity.ExtendedSensor.Path,
    ModulePath := ModulePath, Dir := E_ChannelDir.INPUT);
Ok := _publisher.M_DefineDigitalChannel(NodeIndex := 3, ChannelIndex := RetractedSensorIndex,
    Tag := Identity.RetractedSensor.Tag, DescriptionKey := Identity.RetractedSensor.DescriptionKey,
    Address := Identity.RetractedSensor.Address, Path := Identity.RetractedSensor.Path,
    ModulePath := ModulePath, Dir := E_ChannelDir.INPUT) AND Ok;
Ok := _publisher.M_DefineDigitalChannel(NodeIndex := 4, ChannelIndex := ExtendOutputIndex,
    Tag := Identity.ExtendOutput.Tag, DescriptionKey := Identity.ExtendOutput.DescriptionKey,
    Address := Identity.ExtendOutput.Address, Path := Identity.ExtendOutput.Path,
    ModulePath := ModulePath, Dir := E_ChannelDir.OUTPUT) AND Ok;
Ok := _publisher.M_DefineDigitalChannel(NodeIndex := 4, ChannelIndex := RetractOutputIndex,
    Tag := Identity.RetractOutput.Tag, DescriptionKey := Identity.RetractOutput.DescriptionKey,
    Address := Identity.RetractOutput.Address, Path := Identity.RetractOutput.Path,
    ModulePath := ModulePath, Dir := E_ChannelDir.OUTPUT) AND Ok;
_M_DefineCylinder := Ok;
END_METHOD

END_FUNCTION_BLOCK

// ---- 00_System/FB_PressIoDriver.TcPOU
// Project Hardware Driver layer. This is the only POU that accesses GVL_PressIO.
// It maps raw process-image symbols to semantic HALs and refreshes the Core
// topology publisher. It contains no sequence, mode, recipe or device behavior.
FUNCTION_BLOCK FB_PressIoDriver
VAR
    _publisher : FB_IoTopologyPublisher;
    _unit : REFERENCE TO FB_PressDemoUnit;
    _attached : BOOL;
END_VAR

;

METHOD Setup : BOOL
VAR_INPUT
    UnitRef : REFERENCE TO FB_PressDemoUnit;
END_VAR
_unit REF= UnitRef;
_attached := _publisher.Setup(DataRef := GVL_PressFieldbus.Topology, ResetData := FALSE)
    AND __ISVALIDREF(_unit);
Setup := _attached;
END_METHOD

METHOD M_ReadInputs
VAR_IN_OUT
    PressHal : ST_CylinderHal;
    DoorHal : ST_CylinderHal;
    SlideHal : ST_CylinderHal;
    TwoHandHal : ST_TwoHandHal;
    PowerHal : ST_PowerGroupHal;
    PartPresentHal : ST_DigitalInputHal;
    AirPressureHal : ST_AirPressureHal;
    RawEStopHealthy : BOOL;
    SafeEStopOk : BOOL;
    SafeGuardClosed : BOOL;
    SafeTwoHandActive : BOOL;
    SafePneumaticPermit : BOOL;
    SafetyFieldbusHealthy : BOOL;
    StandardIoHealthy : BOOL;
END_VAR
// Physical feeder retracted = logical slide inside; extended = outside.
SlideHal.ExtendedFb := GVL_PressIO._101B301A;
SlideHal.RetractedFb := GVL_PressIO._101B301B;
DoorHal.ExtendedFb := GVL_PressIO._101B201A;
DoorHal.RetractedFb := GVL_PressIO._101B201B;
PressHal.ExtendedFb := GVL_PressIO._101B202A;
PressHal.RetractedFb := GVL_PressIO._101B202B;
TwoHandHal.RightPressed := GVL_PressIO._101S101;
TwoHandHal.LeftPressed := GVL_PressIO._101S102;
PartPresentHal.Value := GVL_PressIO._101B601;
AirPressureHal.LowPressure := GVL_PressIO._000MB085A_2;
AirPressureHal.OperatingPressure := GVL_PressIO._000MB085A_4;
RawEStopHealthy := GVL_PressIO._000K910A;
PowerHal.PowerFeedback := GVL_PressIO._000K911_Y32;
// Evaluated, fail-closed aliases supplied by TwinSAFE/external safety logic.
SafeEStopOk := GVL_PressSafety._EStopOk;
SafeGuardClosed := GVL_PressSafety._GuardClosed;
SafeTwoHandActive := GVL_PressSafety._TwoHandActive;
SafePneumaticPermit := GVL_PressSafety._PneumaticPermit;
SafetyFieldbusHealthy := GVL_PressSafety._SafetyFieldbusHealthy;
StandardIoHealthy := GVL_PressSafety._StandardIoHealthy;
PartPresentHal.Quality := StandardIoHealthy;
AirPressureHal.Quality := StandardIoHealthy;
END_METHOD

METHOD M_ClearOutputs
GVL_PressIO._101K301A := FALSE; GVL_PressIO._101K301B := FALSE;
GVL_PressIO._101K201A := FALSE; GVL_PressIO._101K201B := FALSE;
GVL_PressIO._101K202A := FALSE; GVL_PressIO._101K202B := FALSE;
GVL_PressIO._101P101 := FALSE; GVL_PressIO._101P102 := FALSE;
GVL_PressIO._000K951_A1 := FALSE; GVL_PressIO._000K911_A1 := FALSE;
END_METHOD

METHOD M_WriteOutputs
VAR_INPUT
    PressHal : ST_CylinderHal;
    DoorHal : ST_CylinderHal;
    SlideHal : ST_CylinderHal;
    PowerHal : ST_PowerGroupHal;
    LampsOn : BOOL;
    ControlCircuitMappingConfirmed : BOOL;
END_VAR
GVL_PressIO._101K301A := SlideHal.ExtendOut;
GVL_PressIO._101K301B := SlideHal.RetractOut;
GVL_PressIO._101K201A := DoorHal.ExtendOut;
GVL_PressIO._101K201B := DoorHal.RetractOut;
GVL_PressIO._101K202A := PressHal.ExtendOut;
GVL_PressIO._101K202B := PressHal.RetractOut;
GVL_PressIO._101P101 := LampsOn;
GVL_PressIO._101P102 := LampsOn;
IF ControlCircuitMappingConfirmed THEN
    GVL_PressIO._000K951_A1 := PowerHal.EnableRequestOut;
    GVL_PressIO._000K911_A1 := PowerHal.EnableRequestOut;
ELSE
    GVL_PressIO._000K951_A1 := FALSE;
    GVL_PressIO._000K911_A1 := FALSE;
END_IF
END_METHOD

METHOD M_RefreshFieldbus
VAR_INPUT
    StandardIoHealthy : BOOL;
END_VAR
VAR
    D : ST_Diagnostic;
END_VAR
IF _attached THEN
    _publisher.M_SetAllHealth(Healthy := StandardIoHealthy);
    _publisher.M_SetDigitalValue(NodeIndex := 3, ChannelIndex := 1, Value := GVL_PressIO._101B301A);
    _publisher.M_SetDigitalValue(NodeIndex := 3, ChannelIndex := 2, Value := GVL_PressIO._101B301B);
    _publisher.M_SetDigitalValue(NodeIndex := 3, ChannelIndex := 3, Value := GVL_PressIO._101B201A);
    _publisher.M_SetDigitalValue(NodeIndex := 3, ChannelIndex := 4, Value := GVL_PressIO._101B201B);
    _publisher.M_SetDigitalValue(NodeIndex := 3, ChannelIndex := 5, Value := GVL_PressIO._101B202A);
    _publisher.M_SetDigitalValue(NodeIndex := 3, ChannelIndex := 6, Value := GVL_PressIO._101B202B);
    _publisher.M_SetDigitalValue(NodeIndex := 3, ChannelIndex := 7, Value := GVL_PressIO._101S101);
    _publisher.M_SetDigitalValue(NodeIndex := 3, ChannelIndex := 8, Value := GVL_PressIO._101S102);
    _publisher.M_SetDigitalValue(NodeIndex := 3, ChannelIndex := 9, Value := GVL_PressIO._000MB085A_2);
    _publisher.M_SetDigitalValue(NodeIndex := 3, ChannelIndex := 10, Value := GVL_PressIO._000MB085A_4);
    _publisher.M_SetDigitalValue(NodeIndex := 3, ChannelIndex := 11, Value := GVL_PressIO._101B601);
    _publisher.M_SetDigitalValue(NodeIndex := 3, ChannelIndex := 12, Value := GVL_PressIO._000K911_Y32);
    _publisher.M_SetDigitalValue(NodeIndex := 3, ChannelIndex := 13, Value := GVL_PressIO._000K910A);
    _publisher.M_SetDigitalValue(NodeIndex := 4, ChannelIndex := 1, Value := GVL_PressIO._101K301A);
    _publisher.M_SetDigitalValue(NodeIndex := 4, ChannelIndex := 2, Value := GVL_PressIO._101K301B);
    _publisher.M_SetDigitalValue(NodeIndex := 4, ChannelIndex := 3, Value := GVL_PressIO._101K201A);
    _publisher.M_SetDigitalValue(NodeIndex := 4, ChannelIndex := 4, Value := GVL_PressIO._101K201B);
    _publisher.M_SetDigitalValue(NodeIndex := 4, ChannelIndex := 5, Value := GVL_PressIO._101K202A);
    _publisher.M_SetDigitalValue(NodeIndex := 4, ChannelIndex := 6, Value := GVL_PressIO._101K202B);
    _publisher.M_SetDigitalValue(NodeIndex := 4, ChannelIndex := 7, Value := GVL_PressIO._101P101);
    _publisher.M_SetDigitalValue(NodeIndex := 4, ChannelIndex := 8, Value := GVL_PressIO._101P102);
    _publisher.M_SetDigitalValue(NodeIndex := 4, ChannelIndex := 9, Value := GVL_PressIO._000K951_A1);
    _publisher.M_SetDigitalValue(NodeIndex := 4, ChannelIndex := 10, Value := GVL_PressIO._000K911_A1);
    _publisher.M_BeginDiagnosticRefresh();
    D := _unit.PressRam.Status.Diagnostic;
    _M_ApplyCylinderDiagnostic(Diagnostic := D,
        ExtendedTag := _unit.PressRam.OutImm.ExtendedSensorTag,
        RetractedTag := _unit.PressRam.OutImm.RetractedSensorTag);
    D := _unit.Door.Status.Diagnostic;
    _M_ApplyCylinderDiagnostic(Diagnostic := D,
        ExtendedTag := _unit.Door.OutImm.ExtendedSensorTag,
        RetractedTag := _unit.Door.OutImm.RetractedSensorTag);
    D := _unit.PartSlide.Status.Diagnostic;
    _M_ApplyCylinderDiagnostic(Diagnostic := D,
        ExtendedTag := _unit.PartSlide.OutImm.ExtendedSensorTag,
        RetractedTag := _unit.PartSlide.OutImm.RetractedSensorTag);
    D := _unit.AirPressureMonitor.Status.Diagnostic;
    _publisher.M_ApplyDiagnostic(Diagnostic := D);
    IF TO_DINT(D.ReasonCode) = PL_ModuleReasons.AIR_SWITCH_CONFLICT THEN
        _publisher.M_ApplyDiagnosticToTag(Diagnostic := D,
            Tag := _unit.AirPressureMonitor.OutImm.LowSensorTag);
        _publisher.M_ApplyDiagnosticToTag(Diagnostic := D,
            Tag := _unit.AirPressureMonitor.OutImm.OperatingSensorTag);
    ELSE
        ;
    END_IF
    _publisher.M_ApplyDiagnostic(Diagnostic := _unit.Status.Diagnostic);
ELSE
    ;
END_IF
END_METHOD

METHOD PRIVATE _M_ApplyCylinderDiagnostic
VAR_INPUT
    Diagnostic : ST_Diagnostic;
    ExtendedTag : STRING(80);
    RetractedTag : STRING(80);
END_VAR
_publisher.M_ApplyDiagnostic(Diagnostic := Diagnostic);
IF TO_DINT(Diagnostic.ReasonCode) = PL_ModuleReasons.CYL_BOTH_SENSORS THEN
    _publisher.M_ApplyDiagnosticToTag(Diagnostic := Diagnostic, Tag := ExtendedTag);
    _publisher.M_ApplyDiagnosticToTag(Diagnostic := Diagnostic, Tag := RetractedTag);
ELSE
    ;
END_IF
END_METHOD

END_FUNCTION_BLOCK

// ---- 00_System/FB_PressControlDomain.TcPOU
// Application control-domain coordinator (Core §9.8). It describes one cage and
// pneumatic power arrangement; it is infrastructure, not a fourth module tier.
FUNCTION_BLOCK FB_PressControlDomain
VAR_OUTPUT
    Status : ST_ControlDomainStatus;
END_VAR
VAR
    _unit : REFERENCE TO FB_PressDemoUnit;
    _attached : BOOL;
END_VAR

;

METHOD Setup : BOOL
VAR_INPUT
    UnitRef : REFERENCE TO FB_PressDemoUnit;
END_VAR
_unit REF= UnitRef;
_attached := __ISVALIDREF(_unit);
Status.Present := TRUE;
Status.Id := 'PRESS-CAGE-01';
Status.Name := 'project.controlDomain.press.name';
Status.MemberCount := 1;
Status.MemberUnitPaths[1] := UnitRef.Name;
Status.Safety.Present := TRUE;
Status.Safety.DeviceCount := 4;
Status.Safety.Devices[1].Present := TRUE;
Status.Safety.Devices[1].Name := 'EStop01';
Status.Safety.Devices[1].Kind := E_SafetyDeviceKind.ESTOP;
Status.Safety.Devices[1].AffectedPowerMask := 16#0000_0001;
Status.Safety.Devices[1].Description := 'project.safety.estopNc';
Status.Safety.Devices[2].Present := TRUE;
Status.Safety.Devices[2].Name := 'PressGuard';
Status.Safety.Devices[2].Kind := E_SafetyDeviceKind.GUARD_DOOR;
Status.Safety.Devices[2].AffectedPowerMask := 16#0000_0001;
Status.Safety.Devices[2].Description := 'project.safety.pressGuard';
Status.Safety.Devices[3].Present := TRUE;
Status.Safety.Devices[3].Name := 'TwoHand01';
Status.Safety.Devices[3].Kind := E_SafetyDeviceKind.TWO_HAND_CONTROL;
Status.Safety.Devices[3].AffectedPowerMask := 16#0000_0001;
Status.Safety.Devices[3].Description := 'project.safety.twoHandControl';
Status.Safety.Devices[4].Present := TRUE;
Status.Safety.Devices[4].Name := 'SafeValve01';
Status.Safety.Devices[4].Kind := E_SafetyDeviceKind.SAFETY_VALVE;
Status.Safety.Devices[4].AffectedPowerMask := 16#0000_0001;
Status.Safety.Devices[4].Description := 'project.safety.pressSafeValve';
Status.ControlPower.Present := TRUE;
Status.ControlPower.GroupCount := 1;
Setup := _attached;
END_METHOD

METHOD M_Update
VAR_INPUT
    SafeEStopOk : BOOL;
    SafeGuardClosed : BOOL;
    SafeTwoHandActive : BOOL;
    SafePneumaticPermit : BOOL;
    SafetyFieldbusHealthy : BOOL;
    StandardIoHealthy : BOOL;
    RawEStopHealthy : BOOL;
    PowerFeedback : BOOL;
    PowerRequested : BOOL;
    TwoHandFieldbusHealthy : BOOL;
END_VAR
IF _attached THEN
    Status.Safety.AllSafe := SafeEStopOk AND SafePneumaticPermit AND SafetyFieldbusHealthy;
    Status.Safety.DemandActive := NOT SafeGuardClosed;
    Status.Safety.ResetRequired := NOT SafeEStopOk;
    Status.Safety.FaultActive := NOT SafetyFieldbusHealthy OR NOT StandardIoHealthy
        OR (RawEStopHealthy <> SafeEStopOk);
    Status.Safety.Devices[1].State := SEL(SafeEStopOk, E_SafetyState.DEMAND, E_SafetyState.READY);
    Status.Safety.Devices[1].Ready := SafeEStopOk;
    Status.Safety.Devices[1].DemandActive := NOT SafeEStopOk;
    Status.Safety.Devices[1].SafeStateActive := NOT SafeEStopOk;
    Status.Safety.Devices[1].ResetRequired := NOT SafeEStopOk;
    Status.Safety.Devices[1].FieldbusHealthy := SafetyFieldbusHealthy;
    Status.Safety.Devices[2].State := SEL(SafeGuardClosed, E_SafetyState.SAFE_STATE, E_SafetyState.READY);
    Status.Safety.Devices[2].Ready := SafeGuardClosed;
    Status.Safety.Devices[2].DemandActive := NOT SafeGuardClosed;
    Status.Safety.Devices[2].SafeStateActive := NOT SafeGuardClosed;
    Status.Safety.Devices[2].FieldbusHealthy := SafetyFieldbusHealthy;
    Status.Safety.Devices[3].State := SEL(SafeTwoHandActive, E_SafetyState.READY, E_SafetyState.DEMAND);
    Status.Safety.Devices[3].Ready := TwoHandFieldbusHealthy;
    Status.Safety.Devices[3].DemandActive := SafeTwoHandActive;
    Status.Safety.Devices[3].SafeStateActive := NOT SafeTwoHandActive;
    Status.Safety.Devices[3].FieldbusHealthy := SafetyFieldbusHealthy;
    Status.Safety.Devices[4].State := SEL(SafePneumaticPermit, E_SafetyState.FAULT, E_SafetyState.READY);
    Status.Safety.Devices[4].Ready := SafePneumaticPermit;
    Status.Safety.Devices[4].DemandActive := NOT SafePneumaticPermit;
    Status.Safety.Devices[4].SafeStateActive := NOT SafePneumaticPermit;
    Status.Safety.Devices[4].FaultActive := NOT SafePneumaticPermit;
    Status.Safety.Devices[4].FieldbusHealthy := SafetyFieldbusHealthy;
    Status.ControlPower.RequestedOn := PowerRequested;
    Status.ControlPower.ControlOn := PowerFeedback;
    Status.ControlPower.Transitioning := _unit.PneumaticPower.Busy;
    Status.ControlPower.RearmRequired := _unit.PneumaticPower.ControlPower.RearmRequired;
    Status.ControlPower.Groups[1] := _unit.PneumaticPower.OutImm.Status;
    Status.ReadyForStart := Status.Safety.AllSafe AND Status.ControlPower.ControlOn
        AND NOT Status.ControlPower.RearmRequired;
ELSE
    Status.ReadyForStart := FALSE;
END_IF
END_METHOD

END_FUNCTION_BLOCK

// ---- 00_System/FB_PressOutputAuthority.TcPOU
// Final ordinary-PLC functional withdrawal layer for the demo. This is defense
// in depth, not a certified safety function; TwinSAFE remains final authority.
FUNCTION_BLOCK FB_PressOutputAuthority

;

METHOD M_Apply
VAR_INPUT
    PowerFeedback : BOOL;
    SafePneumaticPermit : BOOL;
    StandardIoHealthy : BOOL;
    HazardousRamPermit : BOOL;
END_VAR
VAR_IN_OUT
    PressHal : ST_CylinderHal;
    DoorHal : ST_CylinderHal;
    SlideHal : ST_CylinderHal;
END_VAR
IF NOT PowerFeedback OR NOT SafePneumaticPermit OR NOT StandardIoHealthy THEN
    PressHal.ExtendOut := FALSE; PressHal.RetractOut := FALSE;
    DoorHal.ExtendOut := FALSE; DoorHal.RetractOut := FALSE;
    SlideHal.ExtendOut := FALSE; SlideHal.RetractOut := FALSE;
ELSIF NOT HazardousRamPermit THEN
    // Ram-up and assessed low-risk loading actuators remain available.
    PressHal.ExtendOut := FALSE;
ELSE
    ;
END_IF
END_METHOD

END_FUNCTION_BLOCK

// ---- 00_System/FB_PressSimulationDriver.TcPOU
// Simulation Hardware Driver implementing the same semantic HAL boundary as the
// physical driver. No simulation expressions or plant models leak into MAIN.
FUNCTION_BLOCK FB_PressSimulationDriver
VAR
    _pressSim, _doorSim, _slideSim : FB_CylinderSim;
END_VAR

;

METHOD Setup : BOOL
VAR_INPUT
    PressHal : REFERENCE TO ST_CylinderHal;
    DoorHal : REFERENCE TO ST_CylinderHal;
    SlideHal : REFERENCE TO ST_CylinderHal;
END_VAR
_pressSim.Setup(HalRef := PressHal, TravelTime := T#250MS);
_doorSim.Setup(HalRef := DoorHal, TravelTime := T#200MS);
_slideSim.Setup(HalRef := SlideHal, TravelTime := T#300MS);
Setup := TRUE;
END_METHOD

METHOD M_ReadInputs
VAR_INPUT
    SimEStopNc : BOOL;
    SimLeftButton : BOOL;
    SimRightButton : BOOL;
    SimSafetyValveOk : BOOL;
    SimFieldbusHealthy : BOOL;
    SimPartPresent : BOOL;
    SimAirPressureOk : BOOL;
    PowerRequested : BOOL;
END_VAR
VAR_IN_OUT
    DoorHal : ST_CylinderHal;
    TwoHandHal : ST_TwoHandHal;
    PowerHal : ST_PowerGroupHal;
    PartPresentHal : ST_DigitalInputHal;
    AirPressureHal : ST_AirPressureHal;
    RawEStopHealthy : BOOL;
    SafeEStopOk : BOOL;
    SafeGuardClosed : BOOL;
    SafeTwoHandActive : BOOL;
    SafePneumaticPermit : BOOL;
    SafetyFieldbusHealthy : BOOL;
    StandardIoHealthy : BOOL;
END_VAR
// SIMULATION ONLY — these are not safety calculations for a physical machine.
RawEStopHealthy := SimEStopNc;
SafeEStopOk := SimEStopNc AND SimFieldbusHealthy;
SafeGuardClosed := DoorHal.ExtendedFb AND SimFieldbusHealthy;
SafeTwoHandActive := SimLeftButton AND SimRightButton AND SafeEStopOk
    AND SimSafetyValveOk AND SimFieldbusHealthy;
SafePneumaticPermit := SafeEStopOk AND SimSafetyValveOk;
SafetyFieldbusHealthy := SimFieldbusHealthy;
StandardIoHealthy := SimFieldbusHealthy;
PartPresentHal.Value := SimPartPresent;
PartPresentHal.Quality := SimFieldbusHealthy;
AirPressureHal.LowPressure := NOT SimAirPressureOk;
AirPressureHal.OperatingPressure := SimAirPressureOk;
AirPressureHal.Quality := SimFieldbusHealthy;
TwoHandHal.LeftPressed := SimLeftButton;
TwoHandHal.RightPressed := SimRightButton;
PowerHal.PowerFeedback := PowerRequested AND SafePneumaticPermit;
END_METHOD

METHOD M_RefreshPlant
_pressSim();
_doorSim();
_slideSim();
END_METHOD

END_FUNCTION_BLOCK
